// TwinCAT 3 PLC project BX
// ProgramVersion: 3.1.4024.0
// libraries:
//   Tc2_IoFunctions, * (Beckhoff Automation GmbH)
//   Tc2_Math, * (Beckhoff Automation GmbH)
//   Tc2_Standard, * (Beckhoff Automation GmbH)
//   Tc2_System, * (Beckhoff Automation GmbH)
//   Tc2_TcpIp, * (Beckhoff Automation GmbH)
//   Tc2_Utilities, * (Beckhoff Automation GmbH)
//   Tc3_Database, * (Beckhoff Automation GmbH)
//   Tc3_DynamicMemory, * (Beckhoff Automation GmbH)
//   Tc3_EventLogger, * (Beckhoff Automation GmbH)
//   Tc3_JsonXml, * (Beckhoff Automation GmbH)
//   Tc3_Module, * (Beckhoff Automation GmbH)
// project tree:
//   DUTs/00/ DUT_HMI_00.TcDUT, DUT_HMI_00_MANUALS.TcDUT
//   DUTs/01/ DUT_HMI_01.TcDUT, DUT_HMI_01_MANUALS.TcDUT
//   DUTs/02/ DUT_HMI_02.TcDUT, DUT_HMI_02_MANUALS.TcDUT
//   DUTs/03/ DUT_HMI_03.TcDUT, DUT_HMI_03_MANUALS.TcDUT
//   DUTs/04/ DUT_HMI_04.TcDUT, DUT_HMI_04_MANUALS.TcDUT
//   DUTs/05/ DUT_HMI_05.TcDUT, DUT_HMI_05_MANUALS.TcDUT
//   DUTs/06/ DUT_HMI_06.TcDUT, DUT_HMI_06_MANUALS.TcDUT
//   DUTs/07/ DUT_HMI_07.TcDUT, DUT_HMI_07_MANUALS.TcDUT
//   DUTs/08/ DUT_HMI_08.TcDUT, DUT_HMI_08_MANUALS.TcDUT
//   DUTs/09/ DUT_HMI_09.TcDUT, DUT_HMI_09_MANUALS.TcDUT
//   DUTs/10/ DUT_HMI_10.TcDUT, DUT_HMI_10_MANUALS.TcDUT
//   DUTs/11/ DUT_HMI_11.TcDUT, DUT_HMI_11_MANUALS.TcDUT
//   DUTs/12/ DUT_HMI_12.TcDUT, DUT_HMI_12_MANUALS.TcDUT
//   DUTs/13/ DUT_HMI_13.TcDUT, DUT_HMI_13_MANUALS.TcDUT
//   DUTs/14/ DUT_HMI_14.TcDUT, DUT_HMI_14_MANUALS.TcDUT
//   DUTs/15/ DUT_HMI_15.TcDUT, DUT_HMI_15_MANUALS.TcDUT
//   DUTs/16/ DUT_HMI_16.TcDUT, DUT_HMI_16_MANUALS.TcDUT
//   DUTs/Database/ DUT_AppendBatchToProductionQueue.TcDUT, DUT_ChangeBatchPositionInProductionQueue.TcDUT, DUT_CMD_ForceCompletedBatch.TcDUT, DUT_CMD_RecoverBatch.TcDUT, DUT_CMD_RestartBatch.TcDUT, DUT_GetBatchHistory.TcDUT, DUT_GetBatchHistoryDetail.TcDUT, DUT_GetBitting.TcDUT, DUT_CheckCutterAlreadyPresentOnDrums.TcDUT, DUT_GetSettingRepositoryByName.TcDUT, DUT_LogModeStateEvent.TcDUT, DUT_stSPAlarm.TcDUT, DUT_UpdateBroachingProfileSettings.TcDUT, DUT_GetProfilesByFamilyName.TcDUT, DUT_UpdateCuttersOnDrum.TcDUT, DUT_GetResourcesByName.TcDUT, DUT_GetCuttersOnDrum.TcDUT, DUT_NextPartPLCData.TcDUT, DUT_OutInfoOrigin.TcDUT, DUT_ProcessingDataForHMI.TcDUT, DUT_ResourcesByType.TcDUT, DUT_SequenceByName.TcDUT, DUT_SetResourcesByName.TcDUT, DUT_stBroachingPlanBase.TcDUT, DUT_stBatchList.TcDUT, DUT_stBroachingPlanVariants.TcDUT, DUT_stDeleteBatchToProductionQueue.TcDUT, DUT_stExternMarkingData.TcDUT, DUT_stGetPLCData_Buffer.TcDUT, DUT_stMarkingData.TcDUT, DUT_stBroachingPlan.TcDUT, DUT_stOrder.TcDUT, DUT_stOrderItems.TcDUT, DUT_stPLCData.TcDUT, DUT_stProcessingData.TcDUT, DUT_stProcessingHMIData1.TcDUT, DUT_stProcessingHMIData2.TcDUT, DUT_stUpdateBatchToProductionQueue.TcDUT, DUT_UpdateCutterData.TcDUT, DUT_UpdatePartLocationsAndProcessingData.TcDUT, DUT_UpdateSettingRepositoryByName.TcDUT, eDbPiecesStatus.TcDUT
//   DUTs/Database/Mes/ DUT_stMesOrder.TcDUT, DUT_stMesOrderItems.TcDUT
//   DUTs/ DUT_RobSetpoint_Real.TcDUT, DUT_XYZ_Real.TcDUT, DUT_XYZ_Int.TcDUT, eDeviceType.TcTLEO, eLoadingMode.TcDUT, DUT_Events.TcDUT, eBroach.TcDUT, DUT_DataRequest.TcDUT, DUT_MachineData.TcDUT, DUT_MATDiagnostics.TcDUT, DUT_St0Data.TcDUT, DUT_StationData.TcDUT, eConnectionSteps.TcDUT, eEV_Status.TcDUT, eHeaderPieces.TcTLEO, eIcon.TcTLEO, eMode.TcDUT, eProductStatus.TcDUT, eShiftPosMan.TcDUT, eShiftPosPC100.TcDUT, eState.TcTLEO, eStationData.TcDUT, eStationState.TcDUT, stBit.TcDUT, stByteAsBit.TcDUT, stTestStringUnion.TcDUT, stFanucCNCKeyboard.TcDUT, stShiftData.TcDUT, DataBuffer.TcDUT
//   DUTs/EventsMgt/ ST_EventClassInfo.TcDUT, ST_FanucCNCEventAxesMask.TcDUT, ST_FanucCNCEventDetails.TcDUT, ST_FanucCNCEventEntryDetails.TcDUT, ST_FanucCNCEventSourceDetails.TcDUT, ST_FanucCNCEventSourceInfo.TcDUT, ST_FanucCNCEventSourceList.TcDUT, ST_FanucSourceDescriptor.TcDUT, U_FanucCNCEventEntry.TcDUT, U_FanucCNCEventInfo.TcDUT, U_FanucCNCEventSourceInfo.TcDUT
//   DUTs/HMI/ DUT_HIM_ProscessingData.TcDUT, DUT_HIM_DeviceType.TcDUT, DUT_HMI_Display.TcDUT, DUT_HMI_Events.TcDUT, DUT_HMI_EV_Diagnostic.TcDUT, DUT_HMI_EV_Info.TcDUT, DUT_HMI_General.TcDUT, DUT_HMI_General_Manuals.TcDUT, DUT_HMI_Header.TcDUT, DUT_HMI_In.TcDUT, DUT_HMI_In_Resource.TcDUT, DUT_HMI_MesManual.TcDUT, DUT_HMI_Navigation.TcDUT, DUT_HIM_Probe.TcDUT, DUT_HMI_Out.TcDUT, DUT_HMI_Out_Resource.TcDUT, DUT_HMI_Production_Counters.TcDUT, DUT_HMI_Tools.TcDUT, DUT_HMI_UPSStatus.TcDUT
//   DUTs/Production/ DUT_Production.TcDUT, DUT_Production_Counters.TcDUT, DUT_Production_OEE.TcDUT, DUT_Statistics.TcDUT, eOEE.TcDUT
//   FBs/ BytesToWString.TcPOU, FB_ButtonTrigger.TcPOU, FB_DoublingTrigger.TcPOU, FB_LoadingModeChange.TcPOU, FB_OvrMng.TcPOU, FB_PartDataManager.TcPOU, FB_DataBufferManager.TcPOU, FB_PneumaticActuator_2EV.TcPOU, FB_PneumaticActuator_2EV_Diagnostic.TcPOU, FB_Refresh.TcPOU, FB_KillMultipleNavigationPS.TcPOU, FB_RetainTimer.TcPOU, FB_TriggerSequencer.TcPOU, FB_WriteTestFile.TcPOU
//   FBs/Database/FB/ FB_MSSQL_spAppendBatchToProductionQueueFromHMI.TcPOU, FB_MSSQL_spChangeBatchPositionInProductionQueue.TcPOU, FB_MSSQL_spCMD_ForceCompletedBatch.TcPOU, FB_MSSQL_spCMD_HoldBatch.TcPOU, FB_MSSQL_spCMD_RecoverBatch.TcPOU, FB_MSSQL_spCMD_RestartBatch.TcPOU, FB_MSSQL_spCMD_ResumeBatch.TcPOU, FB_MSSQL_spCMD_SuspendBatch.TcPOU, FB_MSSQL_spCMD_UnholdBatch.TcPOU, FB_MSSQL_spDeleteBatchToProductionQueue.TcPOU, FB_MSSQL_spAddProfile.TcPOU, FB_MSSQL_spDeleteCutter.TcPOU, FB_MSSQL_spAddCutter.TcPOU, FB_MSSQL_spGetBatchDetailById.TcPOU, FB_MSSQL_spGetBatchHistory.TcPOU, FB_MSSQL_spGetBatchHistoryByStatus.TcPOU, FB_MSSQL_spGetBatchHistoryDetail.TcPOU, FB_MSSQL_spGetBatchList.TcPOU, FB_MSSQL_spGetBlankKey.TcPOU, FB_MSSQL_spGetBlankKeyByName.TcPOU, FB_MSSQL_spCheckCutterAlreadyPresentOnDrums.TcPOU, FB_MSSQL_spGetCuttersComboboxFormatted.TcPOU, FB_MSSQL_spGetCuttersFromFamilyName.TcPOU, FB_MSSQL_spDeleteProfile.TcPOU, FB_MSSQL_spGetBroachingProfileSettings.TcPOU, FB_MSSQL_spGetSettingRepositoryByName.TcPOU, FB_MSSQL_spUpdateBroachingProfileSettings.TcPOU, FB_MSSQL_spGetProfilesByFamilyName.TcPOU, FB_MSSQL_spGetProfiles.TcPOU, FB_MSSQL_spGetCuttersOnDrum.TcPOU, FB_MSSQL_spGetFamilyNamesForCombobox.TcPOU, FB_MSSQL_spUpdateCuttersOnDrum.TcPOU, FB_MSSQL_spGetCuttersByName.TcPOU, FB_MSSQL_spGetCuttersBySide.TcPOU, FB_MSSQL_spGetCutters.TcPOU, FB_MSSQL_spGetFormattedTablesFromSequences.TcPOU, FB_MSSQL_spGetMillings.TcPOU, FB_MSSQL_spGetMillingsByFamilyName.TcPOU, FB_MSSQL_spGetMillingsByName.TcPOU, FB_MSSQL_spGetOrderInfoList.TcPOU, FB_MSSQL_spGetOrderItems.TcPOU, FB_MSSQL_spGetOrigins.TcPOU, FB_MSSQL_spGetOriginsByName.TcPOU, FB_MSSQL_spGetOriginsBySide.TcPOU, FB_MSSQL_spGetOriginsFromSequence.TcPOU, FB_MSSQL_spGetPartHistory.TcPOU, FB_MSSQL_spGetPartHistoryByBatchName.TcPOU, FB_MSSQL_spGetResourcesByName.TcPOU, FB_MSSQL_spGetResourcesByNameMilling.TcPOU, FB_MSSQL_spGetResourcesByType.TcPOU, FB_MSSQL_spGetResourcesListByType.TcPOU, FB_MSSQL_spGetSettingRepositoryList.TcPOU, FB_MSSQL_spGetSideCode.TcPOU, FB_MSSQL_spSetResourcesByName.TcPOU, FB_MSSQL_spUpdateBatchToProductionQueue.TcPOU, FB_MSSQL_spUpdateCutterData.TcPOU, FB_MSSQL_spUpdateSettingRepositoryByName.TcPOU
//   FBs/Database/FB/Mes/ FB_MSSQL_spMES_GetOrderInfoList.TcPOU, FB_MSSQL_spMES_GetOrderItems.TcPOU
//   FBs/Database/ FB_HMI_SP_Alarm.TcPOU, FB_ProcessingData.TcPOU, PRG_MSSQL_InitConnection.TcPOU, PRG_MSSQL_InitConnection_MyTest1.TcPOU, PRG_MSSQL_InitConnection_MyTest2.TcPOU, PRG_MSSQL_InitConnection_MyTest3.TcPOU, PRG_MSSQL_InitConnection_MyTest4.TcPOU, PRG_MSSQL_InitConnection_MyTest5.TcPOU, PRG_MSSQL_spCMD_AbortProduction.TcPOU, PRG_MSSQL_spMyTest.TcPOU, PRG_MSSQL_spLogModeStateEvent.TcPOU, PRG_MSSQL_spGetNextPartPLCData.TcPOU, PRG_MSSQL_spGetProcessingDataForHMI.TcPOU, PRG_MSSQL_UpdatePartLocationsAndProcessingData.TcPOU
//   FBs/DataRequest/ FB_DataRequest.TcPOU, FC_UnloadManager.TcPOU, FC_BroachingPlanCopyPass.TcPOU, FC_BroachingPlanCopyConpensation.TcPOU, FC_DataFind.TcPOU
//   FBs/Ethernet/ FB_ClientConnection.TcPOU, FB_EthDevice.TcPOU, FB_FrameFifo.TcPOU
//   FBs/Events/ FB_CheckFanucCNCActiveEvents.TcPOU, FB_CheckFanucPMCActiveEvents.TcPOU, FB_PMCEventCollectors.TcPOU, I_EventDetailer.TcIO
//   FBs/LaserMarker - LASIT/ DUT_Job.TcDUT, FB_FlyPowerMarkExeManager.TcPOU, FB_Lasit.TcPOU, FB_LasitManager.TcPOU, FB_FlyPowerMarkManager.TcPOU, FC_Check_ACK.TcPOU, FC_Check_EOT.TcPOU, FC_Check_IN.TcPOU, FC_Check_J.TcPOU, FC_Check_K.TcPOU, FC_Check_R.TcPOU, FC_Check_S.TcPOU, FC_Check_SOH.TcPOU, FC_Check_STX.TcPOU, FC_Check_T.TcPOU
//   FBs/StringBuilder/ clsStringBuilder.TcPOU, I_LimitedStringBuilder.TcIO, I_StringBuilder.TcIO
//   FCs/ FC_AlarmExists.TcPOU, FC_BYTE_TO_BOOLARR.TcPOU, FC_BOOLARR_TO_BYTE.TcPOU, FC_BOOLBYTE_TO_BYTE.TcPOU, FC_BYTE_TO_BOOLBYTE.TcPOU, FC_Concat4.TcPOU, FC_CycleTimeToString.TcPOU, FC_DT_TO_ISO8610.TcPOU, FC_EnumSnakeCaseToString.TcPOU, FC_HeaderCounters.TcPOU, FC_MarkingLayoutSelection.TcPOU, FC_myDTtoString.TcPOU, FC_UpdatePieceCount.TcPOU, FC_OvrManagement.TcPOU, FC_PMCAlarmToBoolArray.TcPOU, FC_PMCWarningToBoolArray.TcPOU, FC_ProductStatus.TcPOU, FC_ProductStatusDatabase.TcPOU, FC_ProductStatusNoPresence.TcPOU, FC_OeeSetUpdateCount.TcPOU, FC_SetPartProgramNameByID.TcPOU, FC_ToBoolArray.TcPOU, FC_ToByte.TcPOU, FC_WIDP_TO_PPNAME.TcPOU, Inc.TcPOU, Print.TcPOU
//   GVLs/ CNC.TcGVL, DB.TcGVL, EC.TcGVL, ETH.TcGVL, G.TcGVL, HMI.TcGVL
//   / PlcTask.TcTTO, ServiceTask.TcTTO
//   POUs/ Database.TcPOU, MAIN.TcPOU, MAIN_SERVICE.TcPOU, PF_00_UPS.TcPOU, PRG_Diagnostic.TcPOU, PRG_EventManagement.TcPOU, PRG_OEE.TcPOU
// real-time tasks:
//   TASK PlcTask: cycle T#1ms, priority 4, ADS port 350
//   TASK ServiceTask: cycle T#50000us, priority 8, ADS port 351
// I/O:
//   DEVICE LAN 1 (EtherCAT), AmsNetId 192.168.159.1.2.1
//     A651 (EP5151-0002) [EP5151-0002 1Ch. Inc. Encoder 24V, M12, single ended]
//     AL671 (CTEU-EtherCAT Modular) [CTEU-EtherCAT Fieldbus modular]
//       modules: Module 1 (VAEM-L1-S-24-PT [48DO])
//     AL673 (CTEU-EtherCAT Modular) [CTEU-EtherCAT Fieldbus modular]
//       modules: Module 1 (VAEM-L1-S-24-PT [48DO])
//   DEVICE LAN 2 (Profinet Device), AmsNetId 192.168.2.200.3.1
//     tcpniodevice [Beckhoff Automation TwinCAT PLC PROFINET I/O Device with I/Os, V2.32, 1 port TwinCAT PN Device]
//       modules: Term 1 (DAP Module), X400 (100 Byte Input), R2000 (200 Byte Input), D2000 (200 Byte Input), Y400 (100 Byte Output), R2200 (200 Byte Output), D2200 (200 Byte Output)
// variable links:
//   BX/BX Instance <-> LAN 1 (EtherCAT)
//     ServiceTask Inputs/EC.EtherCAT_DevState <-> Inputs/DevState
//   BX/BX Instance <-> LAN 1 (EtherCAT)/A651 (EP5151-0002)
//     PlcTask Inputs/EC.I_Ovr_CounterValue <-> ENC Status compact/Counter value
//     PlcTask Inputs/EC.I_Ovr_Overflow <-> ENC Status compact/Status/Counter overflow
//     PlcTask Inputs/EC.I_Ovr_SetCounterDone <-> ENC Status compact/Status/Set counter done
//     PlcTask Inputs/EC.I_Ovr_Underflow <-> ENC Status compact/Status/Counter underflow
//     PlcTask Outputs/EC.Q_Ovr_SetCounter <-> ENC Control compact/Control/Set counter
//     PlcTask Outputs/EC.Q_Ovr_SetCounterValue <-> ENC Control compact/Set counter value
//   BX/BX Instance <-> LAN 1 (EtherCAT)/AL671 (CTEU-EtherCAT Modular)
//     PlcTask Outputs/EC.AL671[{0..4}] <-> Module 1 (VAEM-L1-S-24-PT [48DO])/Outputs/C{1..5} Output  (5 links)
//   BX/BX Instance <-> LAN 1 (EtherCAT)/AL673 (CTEU-EtherCAT Modular)
//     PlcTask Outputs/EC.AL673[{0..5}] <-> Module 1 (VAEM-L1-S-24-PT [48DO])/Outputs/C{1..6} Output  (6 links)
//   BX/BX Instance <-> LAN 2 (Profinet Device)
//     ServiceTask Inputs/EC.ProfiNET_DevState <-> Inputs/DevState
//   BX/BX Instance <-> LAN 2 (Profinet Device)/tcpniodevice
//     PlcTask Inputs/CNC.I_D2200 <-> API/D2200 (200 Byte Output)/Subterm 9 (200 Byte Output)/Inputs/1 Byte Output[0]
//     PlcTask Inputs/CNC.I_D2200 @bit {8..1592 step 8} <-> API/D2200 (200 Byte Output)/Subterm 9 (200 Byte Output)/Inputs/1 Byte Output[{1..199}]  (199 links)
//     PlcTask Inputs/CNC.I_R2200 <-> API/R2200 (200 Byte Output)/Subterm 8 (200 Byte Output)/Inputs/1 Byte Output[0]
//     PlcTask Inputs/CNC.I_R2200 @bit {8..1592 step 8} <-> API/R2200 (200 Byte Output)/Subterm 8 (200 Byte Output)/Inputs/1 Byte Output[{1..199}]  (199 links)
//     PlcTask Inputs/CNC.I_Y400 <-> API/Y400 (100 Byte Output)/Subterm 7 (100 Byte Output)/Inputs/1 Byte Output[0]
//     PlcTask Inputs/CNC.I_Y400 @bit {8..792 step 8} <-> API/Y400 (100 Byte Output)/Subterm 7 (100 Byte Output)/Inputs/1 Byte Output[{1..99}]  (99 links)
//     PlcTask Outputs/CNC.Q_D2000 <-> API/D2000 (200 Byte Input)/Subterm 6 (200 Byte Input)/Outputs/1 Byte Input[0]
//     PlcTask Outputs/CNC.Q_D2000 @bit {8..1592 step 8} <-> API/D2000 (200 Byte Input)/Subterm 6 (200 Byte Input)/Outputs/1 Byte Input[{1..199}]  (199 links)
//     PlcTask Outputs/CNC.Q_R2000 <-> API/R2000 (200 Byte Input)/Subterm 5 (200 Byte Input)/Outputs/1 Byte Input[0]
//     PlcTask Outputs/CNC.Q_R2000 @bit {8..1592 step 8} <-> API/R2000 (200 Byte Input)/Subterm 5 (200 Byte Input)/Outputs/1 Byte Input[{1..199}]  (199 links)
//     ServiceTask Outputs/CNC.Q_X400 <-> API/X400 (100 Byte Input)/Subterm 4 (100 Byte Input)/Outputs/1 Byte Input[0]
//     ServiceTask Outputs/CNC.Q_X400 @bit {8..792 step 8} <-> API/X400 (100 Byte Input)/Subterm 4 (100 Byte Input)/Outputs/1 Byte Input[{1..99}]  (99 links)

CONFIGURATION BX
    RESOURCE PLC ON TwinCAT3
        TASK PlcTask(INTERVAL := T#1ms, PRIORITY := 4);
        TASK ServiceTask(INTERVAL := T#50000us, PRIORITY := 8);
        PROGRAM MAIN WITH PlcTask : MAIN;
        PROGRAM MAIN_SERVICE WITH ServiceTask : MAIN_SERVICE;
    END_RESOURCE
END_CONFIGURATION

// ---- DUTs/00/DUT_HMI_00.TcDUT
TYPE DUT_HMI_00 :
STRUCT
	Manuals 		: DUT_HMI_00_MANUALS;
	EVDiagnostic 	: ARRAY[3..47] OF DUT_HMI_EV_Diagnostic;
	EVInfo			: ARRAY[0..CNC.NUM_MAX_MANUALS_00-1] OF DUT_HMI_EV_Info;
	Status			: USINT;
	CycleTime		: STRING;
END_STRUCT
END_TYPE

// ---- DUTs/00/DUT_HMI_00_MANUALS.TcDUT
TYPE DUT_HMI_00_MANUALS :
STRUCT
	PS : ARRAY[0..CNC.NUM_MAX_MANUALS_00-1] OF BOOL;
	LS : ARRAY[0..CNC.NUM_MAX_MANUALS_00-1] OF BOOL;
END_STRUCT
END_TYPE

// ---- DUTs/01/DUT_HMI_01.TcDUT
TYPE DUT_HMI_01 :
STRUCT
	Manuals 		: DUT_HMI_01_MANUALS;
	ProductStatus 	: eProductStatus;
	State			: eStationState;
	EVDiagnostic 	: ARRAY[0..20] OF DUT_HMI_EV_Diagnostic;
	EVInfo			: ARRAY[0..CNC.NUM_MAX_MANUALS_01-1] OF DUT_HMI_EV_Info;
	Status			: USINT;
	CycleTime		: STRING;
END_STRUCT
END_TYPE

// ---- DUTs/01/DUT_HMI_01_MANUALS.TcDUT
TYPE DUT_HMI_01_MANUALS :
STRUCT
	PS : ARRAY[0..CNC.NUM_MAX_MANUALS_01-1] OF BOOL;
	LS : ARRAY[0..CNC.NUM_MAX_MANUALS_01-1] OF BOOL;
END_STRUCT
END_TYPE

// ---- DUTs/02/DUT_HMI_02.TcDUT
TYPE DUT_HMI_02 :
STRUCT
	Manuals : DUT_HMI_02_MANUALS;
	ProductStatus 	: eProductStatus;
	State			: eStationState;
	EVDiagnostic 	: ARRAY[0..20] OF DUT_HMI_EV_Diagnostic;
	EVInfo			: ARRAY[0..CNC.NUM_MAX_MANUALS_02-1] OF DUT_HMI_EV_Info;
	Status			: USINT;
	CycleTime		: STRING;
END_STRUCT
END_TYPE

// ---- DUTs/02/DUT_HMI_02_MANUALS.TcDUT
TYPE DUT_HMI_02_MANUALS :
STRUCT
	PS : ARRAY[0..CNC.NUM_MAX_MANUALS_02-1] OF BOOL;
	LS : ARRAY[0..CNC.NUM_MAX_MANUALS_02-1] OF BOOL;
END_STRUCT
END_TYPE

// ---- DUTs/03/DUT_HMI_03.TcDUT
TYPE DUT_HMI_03 :
STRUCT
	Manuals : DUT_HMI_03_MANUALS;
	ProductStatus 	: eProductStatus;
	TON_DelayProductStatus : TON;
	RTRIG_ProductStatus : R_TRIG;
	State			: eStationState;
	EVDiagnostic 	: ARRAY[0..20] OF DUT_HMI_EV_Diagnostic;
	EVInfo			: ARRAY[0..CNC.NUM_MAX_MANUALS_03-1] OF DUT_HMI_EV_Info;
	Status			: USINT;
	CycleTime		: STRING;
END_STRUCT
END_TYPE

// ---- DUTs/03/DUT_HMI_03_MANUALS.TcDUT
TYPE DUT_HMI_03_MANUALS :
STRUCT
	PS : ARRAY[0..CNC.NUM_MAX_MANUALS_03-1] OF BOOL;
	LS : ARRAY[0..CNC.NUM_MAX_MANUALS_03-1] OF BOOL;
END_STRUCT
END_TYPE

// ---- DUTs/04/DUT_HMI_04.TcDUT
TYPE DUT_HMI_04 :
STRUCT
	Manuals : DUT_HMI_04_MANUALS;
	ProductStatus 	: eProductStatus;
	State			: eStationState;
	EVDiagnostic 	: ARRAY[0..20] OF DUT_HMI_EV_Diagnostic;
	EVInfo			: ARRAY[0..CNC.NUM_MAX_MANUALS_04-1] OF DUT_HMI_EV_Info;
	Status			: USINT;
	CycleTime		: STRING;
	BroachTarget	: USINT;
END_STRUCT
END_TYPE

// ---- DUTs/04/DUT_HMI_04_MANUALS.TcDUT
TYPE DUT_HMI_04_MANUALS :
STRUCT
	PS : ARRAY[0..CNC.NUM_MAX_MANUALS_04-1] OF BOOL;
	LS : ARRAY[0..CNC.NUM_MAX_MANUALS_04-1] OF BOOL;
END_STRUCT
END_TYPE

// ---- DUTs/05/DUT_HMI_05.TcDUT
TYPE DUT_HMI_05 :
STRUCT
	Manuals : DUT_HMI_05_MANUALS;
	ProductStatus 	: eProductStatus;
	State			: eStationState;
	EVDiagnostic 	: ARRAY[0..20] OF DUT_HMI_EV_Diagnostic;
	EVInfo			: ARRAY[0..CNC.NUM_MAX_MANUALS_05-1] OF DUT_HMI_EV_Info;
	Status			: USINT;
	CycleTime		: STRING;
	BroachTarget	: USINT;
END_STRUCT
END_TYPE

// ---- DUTs/05/DUT_HMI_05_MANUALS.TcDUT
TYPE DUT_HMI_05_MANUALS :
STRUCT
	PS : ARRAY[0..CNC.NUM_MAX_MANUALS_05-1] OF BOOL;
	LS : ARRAY[0..CNC.NUM_MAX_MANUALS_05-1] OF BOOL;
END_STRUCT
END_TYPE

// ---- DUTs/06/DUT_HMI_06.TcDUT
TYPE DUT_HMI_06 :
STRUCT
	Manuals : DUT_HMI_06_MANUALS;
	ProductStatus 	: eProductStatus;
	State			: eStationState;
	EVDiagnostic 	: ARRAY[0..20] OF DUT_HMI_EV_Diagnostic;
	EVInfo			: ARRAY[0..CNC.NUM_MAX_MANUALS_06-1] OF DUT_HMI_EV_Info;
	Status			: USINT;
	CycleTime		: STRING;
	BroachTarget	: USINT;
END_STRUCT
END_TYPE

// ---- DUTs/06/DUT_HMI_06_MANUALS.TcDUT
TYPE DUT_HMI_06_MANUALS :
STRUCT
	PS : ARRAY[0..CNC.NUM_MAX_MANUALS_06-1] OF BOOL;
	LS : ARRAY[0..CNC.NUM_MAX_MANUALS_06-1] OF BOOL;
END_STRUCT
END_TYPE

// ---- DUTs/07/DUT_HMI_07.TcDUT
TYPE DUT_HMI_07 :
STRUCT
	Manuals : DUT_HMI_07_MANUALS;
	ProductStatus 	: eProductStatus;
	State			: eStationState;
	EVDiagnostic 	: ARRAY[0..20] OF DUT_HMI_EV_Diagnostic;
	EVInfo			: ARRAY[0..CNC.NUM_MAX_MANUALS_07-1] OF DUT_HMI_EV_Info;
	Status			: USINT;
	CycleTime		: STRING;
	BroachTarget	: USINT;
END_STRUCT
END_TYPE

// ---- DUTs/07/DUT_HMI_07_MANUALS.TcDUT
TYPE DUT_HMI_07_MANUALS :
STRUCT
	PS : ARRAY[0..CNC.NUM_MAX_MANUALS_07-1] OF BOOL;
	LS : ARRAY[0..CNC.NUM_MAX_MANUALS_07-1] OF BOOL;
END_STRUCT
END_TYPE

// ---- DUTs/08/DUT_HMI_08.TcDUT
TYPE DUT_HMI_08 :
STRUCT
	Manuals : DUT_HMI_08_MANUALS;
	ProductStatus 	: eProductStatus;
	State			: eStationState;
	EVDiagnostic 	: ARRAY[0..20] OF DUT_HMI_EV_Diagnostic;
	EVInfo			: ARRAY[0..CNC.NUM_MAX_MANUALS_08-1] OF DUT_HMI_EV_Info;
	Status			: USINT;
	CycleTime		: STRING;
	BroachTarget	: USINT;
END_STRUCT
END_TYPE

// ---- DUTs/08/DUT_HMI_08_MANUALS.TcDUT
TYPE DUT_HMI_08_MANUALS :
STRUCT
	PS : ARRAY[0..CNC.NUM_MAX_MANUALS_08-1] OF BOOL;
	LS : ARRAY[0..CNC.NUM_MAX_MANUALS_08-1] OF BOOL;
END_STRUCT
END_TYPE

// ---- DUTs/09/DUT_HMI_09.TcDUT
TYPE DUT_HMI_09 :
STRUCT
	Manuals : DUT_HMI_09_MANUALS;
	ProductStatus 	: eProductStatus;
	TON_DelayProductStatus : TON;
	RTRIG_ProductStatus : R_TRIG;
	State			: eStationState;
	EVDiagnostic 	: ARRAY[0..20] OF DUT_HMI_EV_Diagnostic;
	EVInfo			: ARRAY[0..CNC.NUM_MAX_MANUALS_09-1] OF DUT_HMI_EV_Info;
	Status			: USINT;
	CycleTime		: STRING;
	BroachTarget	: USINT;
END_STRUCT
END_TYPE

// ---- DUTs/09/DUT_HMI_09_MANUALS.TcDUT
TYPE DUT_HMI_09_MANUALS :
STRUCT
	PS : ARRAY[0..CNC.NUM_MAX_MANUALS_09-1] OF BOOL;
	LS : ARRAY[0..CNC.NUM_MAX_MANUALS_09-1] OF BOOL;
END_STRUCT
END_TYPE

// ---- DUTs/10/DUT_HMI_10.TcDUT
TYPE DUT_HMI_10 :
STRUCT
	Manuals : DUT_HMI_10_MANUALS;
	ProductStatus 	: eProductStatus;
	State			: eStationState;
	EVDiagnostic 	: ARRAY[0..20] OF DUT_HMI_EV_Diagnostic;
	EVInfo			: ARRAY[0..CNC.NUM_MAX_MANUALS_10-1] OF DUT_HMI_EV_Info;
	Status			: USINT;
	CycleTime		: STRING;
	BroachTarget	: USINT;
END_STRUCT
END_TYPE

// ---- DUTs/10/DUT_HMI_10_MANUALS.TcDUT
TYPE DUT_HMI_10_MANUALS :
STRUCT
	PS : ARRAY[0..CNC.NUM_MAX_MANUALS_10-1] OF BOOL;
	LS : ARRAY[0..CNC.NUM_MAX_MANUALS_10-1] OF BOOL;
END_STRUCT
END_TYPE

// ---- DUTs/11/DUT_HMI_11.TcDUT
TYPE DUT_HMI_11 :
STRUCT
	Manuals : DUT_HMI_11_MANUALS;
	ProductStatus 	: eProductStatus;
	State			: eStationState;
	EVDiagnostic 	: ARRAY[0..20] OF DUT_HMI_EV_Diagnostic;
	EVInfo			: ARRAY[0..CNC.NUM_MAX_MANUALS_11-1] OF DUT_HMI_EV_Info;
	Status			: USINT;
	CycleTime		: STRING;
END_STRUCT
END_TYPE

// ---- DUTs/11/DUT_HMI_11_MANUALS.TcDUT
TYPE DUT_HMI_11_MANUALS :
STRUCT
	PS : ARRAY[0..CNC.NUM_MAX_MANUALS_11-1] OF BOOL;
	LS : ARRAY[0..CNC.NUM_MAX_MANUALS_11-1] OF BOOL;
END_STRUCT
END_TYPE

// ---- DUTs/12/DUT_HMI_12.TcDUT
TYPE DUT_HMI_12 :
STRUCT
	Manuals : DUT_HMI_12_MANUALS;
	ProductStatus 	: eProductStatus;
	State			: eStationState;
	EVDiagnostic 	: ARRAY[0..20] OF DUT_HMI_EV_Diagnostic;
	EVInfo			: ARRAY[0..CNC.NUM_MAX_MANUALS_12-1] OF DUT_HMI_EV_Info;
	Status			: USINT;
	CycleTime		: STRING;
END_STRUCT
END_TYPE

// ---- DUTs/12/DUT_HMI_12_MANUALS.TcDUT
TYPE DUT_HMI_12_MANUALS :
STRUCT
	PS : ARRAY[0..CNC.NUM_MAX_MANUALS_12-1] OF BOOL;
	LS : ARRAY[0..CNC.NUM_MAX_MANUALS_12-1] OF BOOL;
END_STRUCT
END_TYPE

// ---- DUTs/13/DUT_HMI_13.TcDUT
TYPE DUT_HMI_13 :
STRUCT
	Manuals : DUT_HMI_13_MANUALS;
	ProductStatus 	: eProductStatus;
	State			: eStationState;
	EVDiagnostic 	: ARRAY[0..20] OF DUT_HMI_EV_Diagnostic;
	EVInfo			: ARRAY[0..CNC.NUM_MAX_MANUALS_13-1] OF DUT_HMI_EV_Info;
	Status			: USINT;
	CycleTime		: STRING;
END_STRUCT
END_TYPE

// ---- DUTs/13/DUT_HMI_13_MANUALS.TcDUT
TYPE DUT_HMI_13_MANUALS :
STRUCT
	PS : ARRAY[0..CNC.NUM_MAX_MANUALS_13-1] OF BOOL;
	LS : ARRAY[0..CNC.NUM_MAX_MANUALS_13-1] OF BOOL;
END_STRUCT
END_TYPE

// ---- DUTs/14/DUT_HMI_14.TcDUT
TYPE DUT_HMI_14 :
STRUCT
	Manuals : DUT_HMI_14_MANUALS;
	ProductStatus 	: eProductStatus;
	State			: eStationState;
	EVDiagnostic 	: ARRAY[0..20] OF DUT_HMI_EV_Diagnostic;
	EVInfo			: ARRAY[0..CNC.NUM_MAX_MANUALS_14-1] OF DUT_HMI_EV_Info;
	Status			: USINT;
	CycleTime		: STRING;
END_STRUCT
END_TYPE

// ---- DUTs/14/DUT_HMI_14_MANUALS.TcDUT
TYPE DUT_HMI_14_MANUALS :
STRUCT
	PS : ARRAY[0..CNC.NUM_MAX_MANUALS_14-1] OF BOOL;
	LS : ARRAY[0..CNC.NUM_MAX_MANUALS_14-1] OF BOOL;
END_STRUCT
END_TYPE

// ---- DUTs/15/DUT_HMI_15.TcDUT
TYPE DUT_HMI_15 :
STRUCT
	Manuals : DUT_HMI_15_MANUALS;
	ProductStatus 	: eProductStatus;
	State			: eStationState;
	EVDiagnostic 	: ARRAY[0..20] OF DUT_HMI_EV_Diagnostic;
	EVInfo			: ARRAY[0..CNC.NUM_MAX_MANUALS_15-1] OF DUT_HMI_EV_Info;
	Status			: USINT;
	CycleTime		: STRING;
END_STRUCT
END_TYPE

// ---- DUTs/15/DUT_HMI_15_MANUALS.TcDUT
TYPE DUT_HMI_15_MANUALS :
STRUCT
	PS : ARRAY[0..CNC.NUM_MAX_MANUALS_15-1] OF BOOL;
	LS : ARRAY[0..CNC.NUM_MAX_MANUALS_15-1] OF BOOL;
END_STRUCT
END_TYPE

// ---- DUTs/16/DUT_HMI_16.TcDUT
TYPE DUT_HMI_16 :
STRUCT
	Manuals : DUT_HMI_16_MANUALS;
	ProductStatus 	: eProductStatus;
	State			: eStationState;
	EVDiagnostic 	: ARRAY[0..20] OF DUT_HMI_EV_Diagnostic;
	EVInfo			: ARRAY[0..CNC.NUM_MAX_MANUALS_16-1] OF DUT_HMI_EV_Info;
	Status			: USINT;
	CycleTime		: STRING;
END_STRUCT
END_TYPE

// ---- DUTs/16/DUT_HMI_16_MANUALS.TcDUT
TYPE DUT_HMI_16_MANUALS :
STRUCT
	PS : ARRAY[0..CNC.NUM_MAX_MANUALS_16-1] OF BOOL;
	LS : ARRAY[0..CNC.NUM_MAX_MANUALS_16-1] OF BOOL;
END_STRUCT
END_TYPE

// ---- DUTs/Database/DUT_AppendBatchToProductionQueue.TcDUT
TYPE DUT_AppendBatchToProductionQueue :
STRUCT
	return_					: DINT;
	BatchInfoJson			: STRING(DB.MAX_STRING_SIZE);
	BatchItemsJson			: STRING(DB.MAX_STRING_SIZE);
END_STRUCT
END_TYPE

// ---- DUTs/Database/DUT_ChangeBatchPositionInProductionQueue.TcDUT
TYPE DUT_ChangeBatchPositionInProductionQueue:
STRUCT  
	return_value		: DINT;
	BatchId				: STRING(50);
	DestinationPosition : DINT;
END_STRUCT
END_TYPE

// ---- DUTs/Database/DUT_CMD_ForceCompletedBatch.TcDUT
TYPE DUT_CMD_ForceCompletedBatch:
STRUCT  
	return_value	: DINT;
	Id	: STRING(50);
END_STRUCT
END_TYPE

// ---- DUTs/Database/DUT_CMD_RecoverBatch.TcDUT
TYPE DUT_CMD_RecoverBatch:
STRUCT  
	return_value	: DINT;
	Id	: STRING(50);
	Mode	: STRING(50);
END_STRUCT
END_TYPE

// ---- DUTs/Database/DUT_CMD_RestartBatch.TcDUT
TYPE DUT_CMD_RestartBatch:
STRUCT  
	return_value	: DINT;
	Id	: STRING(50);
	Mode	: STRING(50);
	RestartMode	: STRING(50);
END_STRUCT
END_TYPE

// ---- DUTs/Database/DUT_GetBatchHistory.TcDUT
TYPE DUT_GetBatchHistory:
STRUCT  
	return_value	: DINT;
	CurrentPage	: DINT;
	RecordToFetch	: DINT;
END_STRUCT
END_TYPE

// ---- DUTs/Database/DUT_GetBatchHistoryDetail.TcDUT
TYPE DUT_GetBatchHistoryDetail:
STRUCT  
	return_value	: DINT;
	BatchId			: STRING(50);
END_STRUCT
END_TYPE

// ---- DUTs/Database/DUT_GetBitting.TcDUT
TYPE DUT_GetBitting :
STRUCT
	CodeSchema				: STRING(50);
	SideBar					: STRING(50);
END_STRUCT
END_TYPE

// ---- DUTs/Database/DUT_CheckCutterAlreadyPresentOnDrums.TcDUT
TYPE DUT_CheckCutterAlreadyPresentOnDrums :
STRUCT
	Id			: DINT;
	Drum		: STRING(30);
	Present		: DINT;
END_STRUCT
END_TYPE

// ---- DUTs/Database/DUT_GetSettingRepositoryByName.TcDUT
TYPE DUT_GetSettingRepositoryByName:
STRUCT  
	Name		: STRING(50);
	Data		: STRING(DB.MAX_STRING_SIZE);
END_STRUCT
END_TYPE

// ---- DUTs/Database/DUT_LogModeStateEvent.TcDUT
TYPE DUT_LogModeStateEvent :
STRUCT
	return_value 	: DINT;
	EventId			: LINT;
	EventTimeStamp  : DT;
	EventType       : DINT;
	Mode            : DINT;
	State           : DINT;
END_STRUCT
END_TYPE

// ---- DUTs/Database/DUT_stSPAlarm.TcDUT
TYPE DUT_stSPAlarm :
STRUCT
	Error : BOOL;
	ErrorID : DINT;
END_STRUCT
END_TYPE

// ---- DUTs/Database/DUT_UpdateBroachingProfileSettings.TcDUT
TYPE DUT_UpdateBroachingProfileSettings :
STRUCT
	IdBroachingProfileSettings	: DINT;
	DataBroachingProfile		: STRING(DB.MAX_STRING_SIZE);
END_STRUCT
END_TYPE

// ---- DUTs/Database/DUT_GetProfilesByFamilyName.TcDUT
TYPE DUT_GetProfilesByFamilyName :
STRUCT
	FamilyName		: STRING(30);
	JsonResult	: STRING(DB.MAX_STRING_SIZE);
END_STRUCT
END_TYPE

// ---- DUTs/Database/DUT_UpdateCuttersOnDrum.TcDUT
TYPE DUT_UpdateCuttersOnDrum :
STRUCT
	Drum		: STRING(30);
	JsonValue	: STRING(DB.MAX_STRING_SIZE);
END_STRUCT
END_TYPE

// ---- DUTs/Database/DUT_GetResourcesByName.TcDUT
TYPE DUT_GetResourcesByName :
STRUCT
	return_value	: DINT;
	ResourceName	: STRING(50);
END_STRUCT
END_TYPE

// ---- DUTs/Database/DUT_GetCuttersOnDrum.TcDUT
TYPE DUT_GetCuttersOnDrum :
STRUCT
	Drum		: STRING(30);
	JsonResult	: STRING(DB.MAX_STRING_SIZE);
END_STRUCT
END_TYPE

// ---- DUTs/Database/DUT_NextPartPLCData.TcDUT
TYPE DUT_NextPartPLCData :
STRUCT
	return_value: DINT;
	PLCData : STRING(DB.MAX_STRING_SIZE);
END_STRUCT
END_TYPE

// ---- DUTs/Database/DUT_OutInfoOrigin.TcDUT
TYPE DUT_OutInfoOrigin :
STRUCT
	OriginName		: STRING(50);
	NameX			: STRING(10);
	X				: REAL;
	NameY			: STRING(10);
	Y				: REAL;
	NameZ			: STRING(10);
	Z				: REAL;
	NameB			: STRING(10);
	B				: REAL;
END_STRUCT
END_TYPE

// ---- DUTs/Database/DUT_ProcessingDataForHMI.TcDUT
TYPE DUT_ProcessingDataForHMI :
STRUCT
	return_: DINT;
	ProcessingData : STRING(DB.MAX_STRING_SIZE);
END_STRUCT
END_TYPE

// ---- DUTs/Database/DUT_ResourcesByType.TcDUT
TYPE DUT_ResourcesByType :
STRUCT
	return_value	: DINT;
	ReaourceType	: STRING(50);
END_STRUCT
END_TYPE

// ---- DUTs/Database/DUT_SequenceByName.TcDUT
TYPE DUT_SequenceByName :
STRUCT
	return_value	: DINT;
	SequenceName	: STRING(50);
END_STRUCT
END_TYPE

// ---- DUTs/Database/DUT_SetResourcesByName.TcDUT
TYPE DUT_SetResourcesByName :
STRUCT
	return_value	: DINT;
	ReaourceName	: STRING(50);
	NewData			: STRING(DB.MAX_STRING_SIZE);
END_STRUCT
END_TYPE

// ---- DUTs/Database/DUT_stBroachingPlanBase.TcDUT
TYPE DUT_stBroachingPlanBase :
STRUCT
	ToolHolderBase_Position 				: DINT;
	ToolHolderBase_BroachName 			: STRING(50);
	ToolHolderBase_LateralCompensation 	: REAL;
	ToolHolderBase_DepthCompensation 	: REAL;
	ToolHolderBase_AngleCompensation 	: REAL;
END_STRUCT
END_TYPE

// ---- DUTs/Database/DUT_stBatchList.TcDUT
TYPE DUT_stBatchList :
STRUCT
	return_			: DINT;
	InputJson	: STRING(DB.MAX_STRING_SIZE);
	OutputJson	: STRING(DB.MAX_STRING_SIZE);
END_STRUCT
END_TYPE

// ---- DUTs/Database/DUT_stBroachingPlanVariants.TcDUT
TYPE DUT_stBroachingPlanVariants :
STRUCT
   ToolHolderA_Position				: DINT;
   ToolHolderA_BroachName			: STRING(50);
   ToolHolderA_LateralCompensation	: REAL;
   ToolHolderA_DepthCompensation	: REAL;
   ToolHolderA_AngleCompensation	: REAL;
   ToolHolderB_Position				: DINT;
   ToolHolderB_BroachName			: STRING(50);
   ToolHolderB_LateralCompensation	: REAL;
   ToolHolderB_DepthCompensation	: REAL;
   ToolHolderB_AngleCompensation	: REAL;
   ToolHolderC_Position				: DINT;
   ToolHolderC_BroachName			: STRING(50);
   ToolHolderC_LateralCompensation	: REAL;
   ToolHolderC_DepthCompensation	: REAL;
   ToolHolderC_AngleCompensation	: REAL;
   ToolHolderD_Position				: DINT;
   ToolHolderD_BroachName			: STRING(50);
   ToolHolderD_LateralCompensation	: REAL;
   ToolHolderD_DepthCompensation	: REAL;
   ToolHolderD_AngleCompensation	: REAL;
   ToolHolderE_Position				: DINT;
   ToolHolderE_BroachName			: STRING(50);
   ToolHolderE_LateralCompensation	: REAL;
   ToolHolderE_DepthCompensation	: REAL;
   ToolHolderE_AngleCompensation	: REAL;
   ToolHolderF_Position				: DINT;
   ToolHolderF_BroachName			: STRING(50);
   ToolHolderF_LateralCompensation	: REAL;
   ToolHolderF_DepthCompensation	: REAL;
   ToolHolderF_AngleCompensation	: REAL;
END_STRUCT
END_TYPE

// ---- DUTs/Database/DUT_stDeleteBatchToProductionQueue.TcDUT
TYPE DUT_stDeleteBatchToProductionQueue :
STRUCT
	return_			: DINT;
	BatchId	: STRING(50);
END_STRUCT
END_TYPE

// ---- DUTs/Database/DUT_stExternMarkingData.TcDUT
TYPE DUT_stExternMarkingData :
STRUCT
	FrontEnable : ARRAY[0..7] OF BOOL;
	FrontText1 	: STRING(50);
	FrontText2 	: STRING(50);
	FrontText3 	: STRING(50);
	FrontText4 	: STRING(50);
	FrontText5 	: STRING(50);
	FrontText6 	: STRING(50);
	BackEnable 	: ARRAY[0..7] OF BOOL;
	BackText1 	: STRING(50);
	BackText2 	: STRING(50);
	BackText3 	: STRING(50);
	BackText4 	: STRING(50);
	BackText5 	: STRING(50);
	BackText6 	: STRING(50);
END_STRUCT
END_TYPE

// ---- DUTs/Database/DUT_stGetPLCData_Buffer.TcDUT
TYPE DUT_stGetPLCData_Buffer :
STRUCT
	PLCData: STRING(DB.MAX_STRING_SIZE);
END_STRUCT
END_TYPE

// ---- DUTs/Database/DUT_stMarkingData.TcDUT
TYPE DUT_stMarkingData :
STRUCT
    LayoutName 		: STRING(50);
    OrderReference 	: STRING(50);
    ProfileLaser 	: STRING(50);
END_STRUCT
END_TYPE

// ---- DUTs/Database/DUT_stBroachingPlan.TcDUT
TYPE DUT_stBroachingPlan :
STRUCT
    PassCount 		: DINT;
    Pass1BaseBroachingPlan 		: DUT_stBroachingPlanBase;
	Pass1VariantsBroachingPlan 	: DUT_stBroachingPlanVariants;
    Pass2BaseBroachingPlan 		: DUT_stBroachingPlanBase;
	Pass2VariantsBroachingPlan 	: DUT_stBroachingPlanVariants;
    Pass3BaseBroachingPlan 		: DUT_stBroachingPlanBase;
	Pass3VariantsBroachingPlan 	: DUT_stBroachingPlanVariants;
    Pass4BaseBroachingPlan 		: DUT_stBroachingPlanBase;
	Pass4VariantsBroachingPlan 	: DUT_stBroachingPlanVariants;
	Pass5BaseBroachingPlan 		: DUT_stBroachingPlanBase;
	Pass5VariantsBroachingPlan 	: DUT_stBroachingPlanVariants;
END_STRUCT
END_TYPE

// ---- DUTs/Database/DUT_stOrder.TcDUT
TYPE DUT_stOrder :
STRUCT
	Position				: DINT;
	BatchName				: STRING(50);
	Status					: STRING(50);
	ProductName				: STRING(50);
	BlankKeyType			: STRING(10);
	SideBar					: STRING(10);
	Quantity				: DINT;
	ExternMarkingData		: DUT_stExternMarkingData;
	Direct					: BOOL;
END_STRUCT
END_TYPE

// ---- DUTs/Database/DUT_stOrderItems.TcDUT
TYPE DUT_stOrderItems :
STRUCT
	return_			: DINT;
	BatchId	: STRING(50);
END_STRUCT
END_TYPE

// ---- DUTs/Database/DUT_stPLCData.TcDUT
TYPE DUT_stPLCData :
STRUCT
	PartId : DINT;
	RowIndex : STRING(50);
	RunningNo : STRING(50);
  	ProfileName : STRING(50);
  	FamilyName : STRING(50);
  	PlugType : STRING(50);
  	IsFirstPartInBatch : STRING(50);
  	IsLastPartInBatch : STRING(50);
  	IsFirstPartInRow : STRING(50);
  	IsLastPartInRow : STRING(50);
	MarkingData : DUT_stMarkingData;
	Brushing : STRING(50);
	BackHole : STRING(50);
	UnloadingModeId : DINT;
	BroachingPlan : DUT_stBroachingPlan;
END_STRUCT
END_TYPE

// ---- DUTs/Database/DUT_stProcessingData.TcDUT
TYPE DUT_stProcessingData :
STRUCT
	LocationId	: UINT;
	PartId		: LINT;
	StatusId	: eDbPiecesStatus;
	Status		: STRING(10);
	DefectId	: UINT;
	Defect		: STRING;
	ProcessingStartedAt	: STRING(39);
	ProcessingEndedAt	: STRING(39);
	IsInitialUpdate		: STRING(5);
	IsFinalUpdate		: STRING(5);
END_STRUCT
END_TYPE

// ---- DUTs/Database/DUT_stProcessingHMIData1.TcDUT
TYPE DUT_stProcessingHMIData1 :
STRUCT
	LocationId 			: DINT;
	PartId	 			: DINT;
END_STRUCT
END_TYPE

// ---- DUTs/Database/DUT_stProcessingHMIData2.TcDUT
TYPE DUT_stProcessingHMIData2 :
STRUCT
    ProductName 	: STRING(50);
	BatchName 		: STRING(50);
	RowIndex		: STRING(50);
	RowRunningNo    : STRING(50);
	RowQty          : STRING(50);
	OrderReference  : STRING(50);
	Profile         : STRING(50);
	PlugType		: STRING(50);
	Brushing        : STRING(50);
	ProfileLaser    : STRING(50);
	BackHole       	: STRING(50);
    UnloadMode 		: STRING(50);
    RunningNoOverRowQty : STRING(50);
	//CurrentRowOverRowCount  : STRING(50);
END_STRUCT
END_TYPE

// ---- DUTs/Database/DUT_stUpdateBatchToProductionQueue.TcDUT
TYPE DUT_stUpdateBatchToProductionQueue :
STRUCT
	return_			: DINT;
	BatchId	: STRING(DB.MAX_STRING_SIZE);
	BatchInfoJson	: STRING(DB.MAX_STRING_SIZE);
	BatchItemsJson	: STRING(DB.MAX_STRING_SIZE);
END_STRUCT
END_TYPE

// ---- DUTs/Database/DUT_UpdateCutterData.TcDUT
TYPE DUT_UpdateCutterData :
STRUCT
	Id		: DINT;
	Data	: STRING(DB.MAX_STRING_SIZE);
END_STRUCT
END_TYPE

// ---- DUTs/Database/DUT_UpdatePartLocationsAndProcessingData.TcDUT
TYPE DUT_UpdatePartLocationsAndProcessingData :
STRUCT
	return_value	: DINT;
	Data	: STRING(DB.MAX_STRING_SIZE);
END_STRUCT
END_TYPE

// ---- DUTs/Database/DUT_UpdateSettingRepositoryByName.TcDUT
TYPE DUT_UpdateSettingRepositoryByName:
STRUCT  
	return_value	: DINT;
	Name			: STRING(50);
	JsonValue		: STRING(DB.MAX_STRING_SIZE);
END_STRUCT
END_TYPE

// ---- DUTs/Database/eDbPiecesStatus.TcDUT
{attribute 'qualified_only'}
{attribute 'strict'}
TYPE eDbPiecesStatus :
(
	Scrap 		:= -1,
	Undefined	:= 0,
	Fetched		:= 1,
	Processing	:= 2,
	Completed	:= 3
);
END_TYPE

// ---- DUTs/Database/Mes/DUT_stMesOrder.TcDUT
TYPE DUT_stMesOrder :
STRUCT
	return_			: DINT;
	StatusFilter	: STRING(50);
	OrderListJson	: STRING(DB.MAX_STRING_SIZE);
END_STRUCT
END_TYPE

// ---- DUTs/Database/Mes/DUT_stMesOrderItems.TcDUT
TYPE DUT_stMesOrderItems :
STRUCT
	return_			: DINT;
	OrderReference	: STRING(50);
	OrderItemsJson	: STRING(DB.MAX_STRING_SIZE);
END_STRUCT
END_TYPE

// ---- DUTs/DUT_RobSetpoint_Real.TcDUT
TYPE DUT_RobSetpoint_Real :
STRUCT
	Override : USINT;
	PositionOffset : ARRAY[0..EC.NUM_ROBOT_OFFSET - 1] OF DUT_XYZ_Real;
END_STRUCT
END_TYPE

// ---- DUTs/DUT_XYZ_Real.TcDUT
TYPE DUT_XYZ_Real :
STRUCT
	X : REAL;
	Y : REAL;
	Z : REAL;
END_STRUCT
END_TYPE

// ---- DUTs/DUT_XYZ_Int.TcDUT
TYPE DUT_XYZ_Int :
STRUCT
	X : INT;
	Y : INT;
	Z : INT;
END_STRUCT
END_TYPE

// ---- DUTs/eDeviceType.TcTLEO
{attribute 'qualified_only'}
{attribute 'strict'}
TYPE eDeviceType :
(
	Unknown := 0,
	Primary := 1,
	Secondary := 2,
	Remote := 3
);
END_TYPE

// ---- DUTs/eLoadingMode.TcDUT
{attribute 'qualified_only'}
{attribute 'strict'}
TYPE eLoadingMode :
(
	Auto	  := 1,
	Manual	  := 2, 
	SemiAuto  := 3
);
END_TYPE

// ---- DUTs/DUT_Events.TcDUT
TYPE DUT_Events :
STRUCT
	wAlarm						: ARRAY[0..G.MAX_ALR_WORD] OF DWORD;						//Bit mask allarmi
	
	aAlarm						: ARRAY[0..G.MAX_ALR] OF FB_TcAlarm;
	
	Cumulative					: BOOL;
END_STRUCT
END_TYPE

// ---- DUTs/eBroach.TcDUT
{attribute 'qualified_only'}
{attribute 'strict'}
TYPE eBroach :
(
	Master	:= 0,
	V1		:= 2,
	V2		:= 3,
	V3		:= 4,
	V4		:= 5,
	V5		:= 6,
	V6		:= 7
);
END_TYPE

// ---- DUTs/DUT_DataRequest.TcDUT
TYPE DUT_DataRequest :
STRUCT
	aByte	: ARRAY[0..1] OF stByteAsBit; 	
	aDWord	: DWORD;
END_STRUCT
END_TYPE

// ---- DUTs/DUT_MachineData.TcDUT
TYPE DUT_MachineData :
STRUCT
	aBool	: ARRAY[0..79] OF BOOL; 	//10 byte -> 80 bool
	aByte	: ARRAY[0..10] OF USINT;	//10 byte -> 10 usint
	aWord	: ARRAY[0..14] OF UINT;		//60 byte -> 15 uint
	aSt	: ARRAY[1..19] OF DUT_StationData;
END_STRUCT
END_TYPE

// ---- DUTs/DUT_MATDiagnostics.TcDUT
TYPE DUT_MATDiagnostics :
STRUCT
    Running : BOOL;
    Heartbeat : BOOL;
    Error : BOOL;
    ErrorMessage : STRING(80);
END_STRUCT
END_TYPE

// ---- DUTs/DUT_St0Data.TcDUT
TYPE DUT_St0Data :
STRUCT
	FlagP	: ARRAY[0..5] OF BYTE; 	
	RunP	: DWORD;
	WindP	: DWORD;
	NpP		: DWORD;
	Tpcy	: BYTE;
	Tppz	: BYTE;
	TpcyS	: ARRAY[1..48] OF BYTE;
	Data	: ARRAY[1..93] OF DWORD;
	DataB	: ARRAY[1..20] OF BYTE;
	DataAu	: ARRAY[1..10] OF DWORD;
END_STRUCT
END_TYPE

// ---- DUTs/DUT_StationData.TcDUT
TYPE DUT_StationData :
STRUCT
	FlagP_B0 : BYTE;
	FlagP_B1 : BYTE;
	FlagP_B2 : BYTE;
	FlagP_B3 : BYTE;
	FlagP_B4 : BYTE;
	FlagP_B5 : BYTE;
	RunP_B0  : BYTE;
	RunP_B1  : BYTE;
	RunP_B2  : BYTE;
	RunP_B3  : BYTE;
	WidP_B0  : BYTE;
	WidP_B1  : BYTE;
	WidP_B2  : BYTE;
	WidP_B3  : BYTE;
	NppP_B0  : BYTE;
	NppP_B1  : BYTE;
	NppP_B2  : BYTE;
	NppP_B3  : BYTE;
	State    : BYTE;
	Byte_19  : BYTE;		
	Byte_20  : BYTE;		
	Byte_21  : BYTE;		
	Byte_22  : BYTE;		
	Byte_23  : BYTE;		
	Byte_24  : BYTE;		
	Byte_25  : BYTE;		
	Byte_26  : BYTE;		
	Byte_27  : BYTE;		
	Byte_28  : BYTE;		
	Byte_29  : BYTE;		
	Byte_30  : BYTE;		
	Byte_31  : BYTE;		
	Byte_32  : BYTE;		
	Byte_33  : BYTE;		
	Byte_34  : BYTE;		
	Byte_35  : BYTE;		
	Byte_36  : BYTE;		
	Byte_37  : BYTE;		
	Byte_38  : BYTE;		
	Byte_39  : BYTE;		
END_STRUCT
END_TYPE

// ---- DUTs/eConnectionSteps.TcDUT
TYPE eConnectionSteps :
(
	eCONNECTION_STATE_IDLE,
	eCONNECTION_STATE_CONNECT_START,
	eCONNECTION_STATE_CONNECT_WAIT,
	eCONNECTION_STATE_DATAEXCHANGE,
	eCONNECTION_STATE_CLOSE_START,
	eCONNECTION_STATE_CLOSE_WAIT,
	eCONNECTION_STATE_ERROR
);
END_TYPE

// ---- DUTs/eEV_Status.TcDUT
TYPE eEV_Status :
(
	NotUsed								:= -1,
	MovingForward						:= 0,
	MovingBackward						:= 1,
	MoveCompleted						:= 2,
	Timeout								:= 3,
	Error								:= 4
);
END_TYPE

// ---- DUTs/eHeaderPieces.TcTLEO
{attribute 'qualified_only'}
{attribute 'strict'}
TYPE eHeaderPieces :
(
	Ok 		:= 0,
	Ko 		:= 1,
	Loaded	:= 2,
	Total	:= 3,
	End		:= 4
);
END_TYPE

// ---- DUTs/eIcon.TcTLEO
{attribute 'qualified_only'}
{attribute 'strict'}
TYPE eIcon :
(
	Emg			:= 0,
	DoorOpen	:= 1,
	AirOk		:= 2,
	HydraulicOk	:= 3,
	EquipmentOk	:= 4,
	Home		:= 5,
	Connection	:= 6,
	End			:= 16
);
END_TYPE

// ---- DUTs/eMode.TcDUT
{attribute 'qualified_only'}
{attribute 'strict'}
TYPE eMode :
(
	MODE_MANUAL := 0,
	MODE_SINGLE := 1,
	MODE_AUTO := 2,
	MODE_MAINTENANCE := 3
);
END_TYPE

// ---- DUTs/eProductStatus.TcDUT
{attribute 'qualified_only'}
{attribute 'strict'}
TYPE eProductStatus :
(
	Scraped 	:= -1,
	NotPresent 	:= 0,
	Present 	:= 1,
	Working 	:= 2,
	Completed 	:= 3
);
END_TYPE

// ---- DUTs/eShiftPosMan.TcDUT
{attribute 'qualified_only'}
{attribute 'strict'}
TYPE eShiftPosMan :
(
	eSt0 := 0,
	eSt1 := 1,
	eSt2 := 2,
	eSt3 := 3,
	eSt4 := 4,
	eSt5 := 5,
	eSt6 := 6,
	eSt7 := 7,
	eSt8 := 8,
	eSt9 := 9,
	eSt10 := 10,
	eSt11 := 11,
	eSt12 := 12,
	eSt13 := 13,
	eSt14 := 14,
	eSt15 := 15,
	eSt16 := 16,
	eSt17 := 17,
	eSt18 := 18,
	eSt19 := 19,
	eSt20 := 20
);
END_TYPE

// ---- DUTs/eShiftPosPC100.TcDUT
{attribute 'qualified_only'}
{attribute 'strict'}
TYPE eShiftPosPC100 :
(
	eSt2b := 0,
	eSt2c := 1,
	eSt2d := 2
);
END_TYPE

// ---- DUTs/eState.TcTLEO
{attribute 'qualified_only'}
{attribute 'strict'}
TYPE eState :
(
	Undefine	:= -1,
	PowerOff	:= 0,
	Home		:= 1,
	Ready		:= 2,
	Running		:= 3,
	Alarm		:= 4,
	Emptying	:= 5,
	Loading		:= 6,
	Manual		:= 7,
	UpsOn		:= 99 //solo per database, creato internamente in PLC Beckhoff
);
END_TYPE
//  Undefine = '-1'

// ---- DUTs/eStationData.TcDUT
{attribute 'qualified_only'}
{attribute 'strict'}
TYPE eStationData :
(
	aSt1	:= 0,
	aSt2	:= 1,
	aSt3	:= 2,
	aSt4	:= 3,
	aSt5	:= 4,
	aSt6	:= 5,
	aSt7	:= 6,
	aSt8	:= 7,
	aSt9	:= 8,
	aSt10	:= 9,
	aSt11	:= 10,
	aSt12	:= 11,
	aSt13	:= 12,
	aSt14	:= 13,
	aSt15	:= 14,
	aSt16	:= 15,
	aSt2b	:= 16,
	aSt2c	:= 17,
	aSt2d	:= 18
);
END_TYPE

// ---- DUTs/eStationState.TcDUT
{attribute 'qualified_only'}
{attribute 'strict'}
TYPE eStationState :
(
	Alarm 		:= -1,
	Disable 	:= 0,
	Ready 		:= 1,
	Working		:= 2,
	EndOfJob	:= 3,
	Undefine	:= 4,
	Extraction	:= 5,
	Infeed		:= 6
);
END_TYPE

// ---- DUTs/EventsMgt/ST_EventClassInfo.TcDUT
TYPE ST_EventClassInfo :
STRUCT
	GUID : GUID;
	BaseAddress : POINTER TO TcEventEntry;
	Count : UDINT;
END_STRUCT
END_TYPE

// ---- DUTs/EventsMgt/ST_FanucCNCEventAxesMask.TcDUT
TYPE ST_FanucCNCEventAxesMask :
STRUCT
	Axis_1 : BIT;
	Axis_2 : BIT;
	Axis_3 : BIT;
	Axis_4 : BIT;
	Axis_5 : BIT;
	Axis_6 : BIT;
	Axis_7 : BIT;
	Axis_8 : BIT;
END_STRUCT
END_TYPE

// ---- DUTs/EventsMgt/ST_FanucCNCEventDetails.TcDUT
TYPE ST_FanucCNCEventDetails :
STRUCT
	AxesMask : ST_FanucCNCEventAxesMask;
	Category : BYTE;
	No : UINT;
END_STRUCT
END_TYPE

// ---- DUTs/EventsMgt/ST_FanucCNCEventEntryDetails.TcDUT
TYPE ST_FanucCNCEventEntryDetails :
STRUCT
	SourceInfo : U_FanucCNCEventSourceInfo;
	EventInfo : U_FanucCNCEventInfo;
END_STRUCT
END_TYPE

// ---- DUTs/EventsMgt/ST_FanucCNCEventSourceDetails.TcDUT
TYPE ST_FanucCNCEventSourceDetails :
STRUCT
	MainType : BYTE;
	SubType : BYTE;
	CNCNo : BYTE;
	PathNo : BYTE;
END_STRUCT
END_TYPE

// ---- DUTs/EventsMgt/ST_FanucCNCEventSourceInfo.TcDUT
TYPE ST_FanucCNCEventSourceInfo :
STRUCT
	SourceId : U_FanucCNCEventSourceInfo;		// 4 bytes					=  4
	CNCName : STRING[21];						// (21 + 1) bytes			= 22
	PathName : STRING[21];						// (21 + 1) bytes			= 22
	AxisNames : ARRAY [1..8] OF STRING[3];		// 8 * (3 + 1) = 32 bytes	= 32
END_STRUCT										//					Totale	= 80
END_TYPE

// ---- DUTs/EventsMgt/ST_FanucCNCEventSourceList.TcDUT
TYPE ST_FanucCNCEventSourceList :
STRUCT
	FanucCNCSources : ARRAY [1..NUM_MAX_CNC_EVENT_SOURCES] OF ST_FanucCNCEventSourceInfo;
	HashMD5 : ARRAY[0..15] OF BYTE;
END_STRUCT
END_TYPE

// ---- DUTs/EventsMgt/ST_FanucSourceDescriptor.TcDUT
TYPE ST_FanucSourceDescriptor :
STRUCT
	MainType : BYTE;
	SubType : BYTE;
	CNCNo : BYTE;
	PathNo : BYTE;
END_STRUCT
END_TYPE

// ---- DUTs/EventsMgt/U_FanucCNCEventEntry.TcDUT
TYPE U_FanucCNCEventEntry :
UNION
	{attribute 'displaymode':='hex'}
	Id : LWORD;
	Details : ST_FanucCNCEventEntryDetails;	
END_UNION
END_TYPE

// ---- DUTs/EventsMgt/U_FanucCNCEventInfo.TcDUT
TYPE U_FanucCNCEventInfo :
UNION
	{attribute 'displaymode':='hex'}
	Id : WORD;
	Details : ST_FanucCNCEventDetails;
END_UNION

END_TYPE

// ---- DUTs/EventsMgt/U_FanucCNCEventSourceInfo.TcDUT
TYPE U_FanucCNCEventSourceInfo :
UNION
	{attribute 'displaymode':='hex'}
	Id : DWORD;
	Details : ST_FanucCNCEventSourceDetails;
END_UNION

END_TYPE

// ---- DUTs/HMI/DUT_HIM_ProscessingData.TcDUT
TYPE DUT_HIM_ProscessingData :
STRUCT
	Name			: STRING(10);
	PartId			: DINT;
    ProductName 	: STRING(50);
	BatchName 		: STRING(50);
	RowIndex		: STRING(50);
	RowRunningNo    : STRING(50);
	RowQty          : STRING(50);
	OrderReference  : STRING(50);
	Profile 		: STRING(50);
	PlugType       	: STRING(50);
	Brushing     	: STRING(50);
	ProfileLaser    : STRING(50);
	BackHole        : STRING(50);
	UnloadMode      : STRING(50);
    RunningNoOverRowQty : STRING(50);
	CurrentRowOverRowCount  : STRING(50);	
	ProductStatus			: eProductStatus;
END_STRUCT
END_TYPE

// ---- DUTs/HMI/DUT_HIM_DeviceType.TcDUT
TYPE DUT_HIM_DeviceType :
STRUCT
	Ip : STRING(15);
	DeviceType : eDeviceType;
END_STRUCT
END_TYPE

// ---- DUTs/HMI/DUT_HMI_Display.TcDUT
TYPE DUT_HMI_Display :
STRUCT
	Enable: BOOL;
	Value:DINT;
END_STRUCT
END_TYPE

// ---- DUTs/HMI/DUT_HMI_Events.TcDUT
TYPE DUT_HMI_Events :
STRUCT
	Clear :BOOL;
END_STRUCT
END_TYPE

// ---- DUTs/HMI/DUT_HMI_EV_Diagnostic.TcDUT
TYPE DUT_HMI_EV_Diagnostic :
STRUCT
	Enable	 : BOOL;
	dFwdTime : UINT;
	dBwdTime : UINT;
	eStatus  : eEV_Status;
	Error 	 : BOOL;	
END_STRUCT
END_TYPE

// ---- DUTs/HMI/DUT_HMI_EV_Info.TcDUT
TYPE DUT_HMI_EV_Info :
STRUCT
	Enable	 : BOOL;
	dTime 	 : UINT;
	Error 	 : BOOL;	
END_STRUCT
END_TYPE

// ---- DUTs/HMI/DUT_HMI_General.TcDUT
TYPE DUT_HMI_General :
STRUCT
	Manuals 	: DUT_HMI_General_Manuals;		// Fanuc 
	Mes			: DUT_HMI_MesManual;
END_STRUCT
END_TYPE

// ---- DUTs/HMI/DUT_HMI_General_Manuals.TcDUT
TYPE DUT_HMI_General_Manuals :
STRUCT
	PS : ARRAY[0..CNC.NUM_MAX_MANUALS_GENERAL-1] OF BOOL;
	LS : ARRAY[0..CNC.NUM_MAX_MANUALS_GENERAL-1] OF BOOL;
END_STRUCT
END_TYPE

// ---- DUTs/HMI/DUT_HMI_Header.TcDUT
TYPE DUT_HMI_Header :
STRUCT
	OperatingMode	: eMode;
	MachineState	: eState;
	Override 		: STRING(3);
	OvrMultiplier	: STRING(3);
	OvrMultFeedback	: BOOL;
	Feedrate 		: STRING(3);
	Icons			: ARRAY[0..eIcon.End] OF BOOL;
	Equipment 		: STRING;
	Pieces			: ARRAY[0..eHeaderPieces.End] OF UDINT;
	ProgressBar		: USINT;
	PathActive		: STRING(2);
END_STRUCT
END_TYPE

// ---- DUTs/HMI/DUT_HMI_In.TcDUT
TYPE DUT_HMI_In :
STRUCT
	AxisSelected 		: USINT;
	Tools				: DUT_HMI_Tools;
	Header				: DUT_HMI_Header;
	Events				: DUT_HMI_Events;
	Navigation			: DUT_HMI_Navigation;
	Dummy				: ARRAY[0..9] OF BOOL; // Non ho capito perchè ma in qualche modo pannelo scrive più memoria oltre in navigation, quindi ho dichiarato questa variabile
												// per occupare memoria a caso, se no pannello mi tenva forzata la roba di statistics
	Statistics			: DUT_Statistics;
	Resource			: DUT_HMI_In_Resource;
	LoadingModeChanged  : BOOL;
END_STRUCT
END_TYPE

// ---- DUTs/HMI/DUT_HMI_In_Resource.TcDUT
TYPE DUT_HMI_In_Resource :
STRUCT
	ProductName		: STRING(50);
	Refresh			: BOOL;
END_STRUCT
END_TYPE

// ---- DUTs/HMI/DUT_HMI_MesManual.TcDUT
TYPE DUT_HMI_MesManual :
STRUCT
	PS : BOOL;
	LS : BOOL;
	Data : STRING(DB.MAX_STRING_SIZE);
END_STRUCT
END_TYPE

// ---- DUTs/HMI/DUT_HMI_Navigation.TcDUT
TYPE DUT_HMI_Navigation :
STRUCT
	PS : ARRAY[0..HMI.NUM_NAVIGATION_ITEMS-1] OF BOOL;
	LS : ARRAY[0..HMI.NUM_NAVIGATION_ITEMS-1] OF BOOL;
END_STRUCT
END_TYPE

// ---- DUTs/HMI/DUT_HIM_Probe.TcDUT
TYPE DUT_HIM_Probe :
STRUCT
	ActualProbeValue : REAL;
	ActualEncoderValue : REAL;
	Error	: BOOL;
	UpperLimit	: REAL;
	LowerLimit	: REAL;
END_STRUCT
END_TYPE

// ---- DUTs/HMI/DUT_HMI_Out.TcDUT
TYPE DUT_HMI_Out :
STRUCT
	UPSDiagnostic 	: DUT_HMI_UPSStatus;
	Header		  	: DUT_HMI_Header;
	AxisSelected  	: USINT;
	Tools			: DUT_HMI_Tools;
	OrderList 		: ARRAY[0..G.PRODUCTIONTABLE_SIZE] OF DUT_stOrder;
	Doors			: ARRAY[0..5] OF SINT;
	Gc1000Status	: SINT;
	Resource		: DUT_HMI_Out_Resource;
	Probe			: DUT_HIM_Probe;
	CycleTime		: STRING(50);
	Counters		: DUT_HMI_Production_Counters;
	ProductionQueueRefresh : BOOL;
	KebaEnabled	: BOOL;
	KebaHMILoaded : BOOL;
	IpDevices	: ARRAY[0..1] OF DUT_HIM_DeviceType;
	EnableProductionAction: BOOL;
	ResfreshPermissions : BOOL;
END_STRUCT
END_TYPE

// ---- DUTs/HMI/DUT_HMI_Out_Resource.TcDUT
TYPE DUT_HMI_Out_Resource :
STRUCT
	Origin : DUT_OutInfoOrigin;
END_STRUCT
END_TYPE

// ---- DUTs/HMI/DUT_HMI_Production_Counters.TcDUT
TYPE DUT_HMI_Production_Counters :
STRUCT
	TotalPieceGood : UDINT;
	TotalPieceScrap : UDINT;
END_STRUCT
END_TYPE

// ---- DUTs/HMI/DUT_HMI_Tools.TcDUT
TYPE DUT_HMI_Tools :
STRUCT
	TaskManager			: BOOL; // Open Windows Task Manager program
	CNCScreenDisplay 	: BOOL; // Open Fancu CNC Screen Display program
	ProgramTransferTool : BOOL; // Open Fanuc Program Transfer Tool program
	OnScreenKeyboard	: BOOL; // Open On Screen Kryboard tool
	CloseBrowser		: BOOL; // Close browser and HMI application
	FanucLadder			: BOOL; // Open Fanuc Ladder program
	FlyCad				: BOOL; // Open Lasit FlyCad software
	OpenPage			: BOOL; // Open tools page
END_STRUCT
END_TYPE

// ---- DUTs/HMI/DUT_HMI_UPSStatus.TcDUT
TYPE DUT_HMI_UPSStatus :
STRUCT
	Valid : BOOL;
	State : ST_UPSStatus;
END_STRUCT
END_TYPE

// ---- DUTs/Production/DUT_Production.TcDUT
TYPE DUT_Production :
STRUCT
	Counters				: DUT_Production_Counters; // Piece Counters
	OEE						: DUT_Production_OEE; // OEE Parameters
END_STRUCT
END_TYPE

// ---- DUTs/Production/DUT_Production_Counters.TcDUT
TYPE DUT_Production_Counters :
STRUCT
	TotalPieces						: UDINT; 	// Contatore totale pezzi
	PartialPieces					: UDINT; 	// Contatore pezzi resettabile manualmente
	PartialActualGood				: UDINT;	// COntatore pezzi buoni resettabile manualmente
	BatchPieces						: UDINT;	// Pezzi da produrre per il lotto
	ActualGood						: UDINT;	// Pezzi ok
	ActualPieces					: DINT;		// Pezzi già prodotti per il lotto
	ActualScrap						: DINT;		// Pezzi già prodotti per il lotto
	PiecesPerHour 					: ARRAY[0..23] OF REAL;
	MaxPiecesPerHour 				: REAL;
	ActualDate						: ARRAY [0..2] OF WORD;
	ActivePiecesDaily_PreviousHours	: REAL;
	Pieces_Daily					: REAL;
	BatchPiecesUpdateConfirm		: BOOL;
	BatchPiecesUpdateAbort			: BOOL;
	BatchPiecesTextInputValue		: UDINT;
END_STRUCT
END_TYPE

// ---- DUTs/Production/DUT_Production_OEE.TcDUT
TYPE DUT_Production_OEE :
STRUCT
	Availabilty 			: REAL;
	Performance 			: REAL;
	Quality					: REAL;
	tON						: REAL; // Tempo di reale produzione in Production Mode
	tOFF					: REAL; // Tempo di attesa operatore in Production Mode
	tDOWN					: REAL; // Tempo di macchina in uno stato che non può produrre
	s_tON					: STRING; // Tempo di reale produzione in Production Mode
	s_tOFF					: STRING; // Tempo di attesa operatore in Production Mode
	s_tDOWN					: STRING; // Tempo di macchina in uno stato che non può produrre
	s_tTOTAL				: STRING; // Tempo di osservazione
	OEE						: REAL;
	GoodPieces				: DINT;
	BadPieces				: DINT;
	IdealCycleTime			: TIME := T#9s;
	PlannedProductionTime	: DWORD := 60;
	OperatingTime			: TIME;
END_STRUCT
END_TYPE

// ---- DUTs/Production/DUT_Statistics.TcDUT
TYPE DUT_Statistics :
STRUCT
	OEE_Enable				: BOOL;
	OEE_Reset				: BOOL;
END_STRUCT
END_TYPE

// ---- DUTs/Production/eOEE.TcDUT
{attribute 'qualified_only'}
{attribute 'strict'}
TYPE eOEE :
(
	Downtime 	:= 0,
	Uptime	 	:= 1,
	Pause		:= 2,
	Completed	:= 3
);
END_TYPE

// ---- DUTs/stBit.TcDUT
TYPE stBit :
STRUCT
    b0  : BIT;
    b1  : BIT;
    b2  : BIT;
    b3  : BIT;
    b4  : BIT;
    b5  : BIT;
    b6  : BIT;
    b7  : BIT; 
END_STRUCT
END_TYPE

// ---- DUTs/stByteAsBit.TcDUT
TYPE stByteAsBit :
UNION
	aByte	: BYTE;
	aBit	: stBit;
END_UNION
END_TYPE

// ---- DUTs/stTestStringUnion.TcDUT
TYPE stTestStringUnion :
UNION
	sString		: STRING(DB.MAX_STRING_SIZE);
	nByte		: ARRAY[0..DB.MAX_STRING_SIZE] OF BYTE;
END_UNION
END_TYPE

// ---- DUTs/stFanucCNCKeyboard.TcDUT
TYPE stFanucCNCKeyboard :
STRUCT
	PS: ARRAY[0..(NUM_MAX_CNC_KEYBOARD_FOR_BECKHOFF-1)] OF BOOL;
	LS: ARRAY[0..(NUM_MAX_CNC_KEYBOARD_FOR_BECKHOFF-1)] OF BOOL;
END_STRUCT
END_TYPE

// ---- DUTs/stShiftData.TcDUT
TYPE stShiftData :
STRUCT
	FLAGP : stByteAsBit;
	WIDP : DINT;
	
	PmcData : DUT_St0Data;
	stPLCData 			: DUT_stPLCData;
	ProcessingData 		: DUT_stProcessingHMIData2;
END_STRUCT
END_TYPE

// ---- DUTs/DataBuffer.TcDUT
TYPE DataBuffer :
STRUCT
	WIDP : DINT;
	PmcData : DUT_St0Data;
	stPLCData 			: DUT_stPLCData;
END_STRUCT
END_TYPE

// ---- FBs/LaserMarker - LASIT/DUT_Job.TcDUT
TYPE DUT_Job :
STRUCT
	JobName			: STRING(50);
	JobIndex		: USINT;
	IndexDynamicCmd	: ARRAY[1..10] OF BOOL;
END_STRUCT
END_TYPE

// ---- GVLs/CNC.TcGVL
VAR_GLOBAL CONSTANT
// Events
	NUM_CNC_EVENTS 					: UINT := 5000;	
	NUM_PMC_EVENTS 					: UINT := 4000;
	NUM_MAX_CNC_ACTIVE_EVENTS 		: UINT := 50;
	NUM_MAX_CNC_EVENT_SOURCES 		: UINT := 50;
	NUM_MAX_STATION_ALARMS			: UINT := 80;
	NUM_MAX_STATION_WARNINGS		: UINT := 16;
	NUM_MAX_GENERAL_ALARMS			: UINT := 160;
	NUM_MAX_GENERAL_WARNINGS		: UINT := 200;
	NUM_00_ALARMS					: UINT := 300;
	NUM_00_WARNINGS					: UINT := 100;
	
// Navigation
	NUM_NAVIGATION_ITEMS 			: UINT := 3;	// Numero di byte scritti su pmc
	
// Keyboard layout	
	NUM_MAX_CNC_KEYBOARD_FOR_BECKHOFF 	: UINT := 64;
	NUM_MAX_CNC_KEYBOARD			: UINT := 8;

// Buttons and leds	
	NUM_MAX_CNC_BUTTONS_LEDS  		: UINT := 500;
	
// HS
	NUM_HS_EACH_STATION				: UINT := 50;
	
// Number of stations
	NUM_STATIONS					: UINT := 9;
	NUM_DATA_POSITION				: UINT := 14;
	
	NUM_MAX_MANUALS_GENERAL 		: UINT := 480;
	NUM_MAX_MANUALS_00 				: UINT := 320;
	NUM_MAX_MANUALS_01 				: UINT := 80;
	NUM_MAX_MANUALS_02 				: UINT := 80;
	NUM_MAX_MANUALS_03 				: UINT := 80;
	NUM_MAX_MANUALS_04 				: UINT := 80;
	NUM_MAX_MANUALS_05 				: UINT := 80;
	NUM_MAX_MANUALS_06 				: UINT := 80;
	NUM_MAX_MANUALS_07 				: UINT := 80;
	NUM_MAX_MANUALS_08 				: UINT := 80;
	NUM_MAX_MANUALS_09 				: UINT := 80;
	NUM_MAX_MANUALS_10 				: UINT := 80;
	NUM_MAX_MANUALS_11 				: UINT := 80;
	NUM_MAX_MANUALS_12 				: UINT := 80;
	NUM_MAX_MANUALS_13 				: UINT := 80;
	NUM_MAX_MANUALS_14 				: UINT := 80;
	NUM_MAX_MANUALS_15 				: UINT := 80;
	NUM_MAX_MANUALS_16 				: UINT := 80;
	NUM_MAX_MANUALS_17 				: UINT := 80;
	NUM_MAX_MANUALS_18 				: UINT := 80;
	
	IPAddress						: STRING := '192.168.1.1';
END_VAR

{attribute 'qualified_only'}
VAR_GLOBAL
	vKeyboard : stFanucCNCKeyboard;
	MachineData	: DUT_MachineData;
	MachineStatus : ARRAY[1..4] OF USINT;
	DataRequestRead : DUT_DataRequest;
	DataRequestWrite : DUT_DataRequest;
	
// MAT - Data exchange FOCAS-ADS
// vKeyboard	
	Q_R3900 AT %MB3000 	: ARRAY[0..(NUM_MAX_CNC_KEYBOARD-1)] OF BYTE; // vKeyboard - Keys Area 
	MATDiagnostic_MB3000 : DUT_MATDiagnostics;
	I_R3950 AT %MB3500 	: ARRAY[0..(NUM_MAX_CNC_KEYBOARD-1)] OF BYTE; // vKeyboard - Leds Area 
	MATDiagnostic_MB3500 : DUT_MATDiagnostics;
	
// Buttons/Leds
	Q_R4000 AT %MB14000 : ARRAY[0..(NUM_MAX_CNC_BUTTONS_LEDS-1)] OF BYTE; // Buttons
	MATDiagnostic_MB14000 : DUT_MATDiagnostics;
	I_R4500 AT %MB14500 : ARRAY[0..(NUM_MAX_CNC_BUTTONS_LEDS-1)] OF BYTE; // Leds
	MATDiagnostic_MB14500 : DUT_MATDiagnostics;
			
// MachineData
	I_E0000 AT %MB8000 : ARRAY[0..1999] OF BYTE;
	MATDiagnostic_MB8000 : DUT_MATDiagnostics;
	
// St0 Data
	St0Data AT %MB20000 : ARRAY[0..499] OF BYTE;
	St0DataTemp : DUT_St0Data;
	MATDiagnostic_MB20000 : DUT_MATDiagnostics;
	
// HS_write
	HS_write AT %MB4000 : ARRAY[0..12] OF BYTE;
	MATDiagnostic_MB4000 : DUT_MATDiagnostics;	

// HS_read
	HS_read AT %MB6000 : ARRAY[0..9] OF BYTE;
	MATDiagnostic_MB6000 : DUT_MATDiagnostics;
	
// FlyPowerOn // scritto da MatManager
	FlyPowerMarkOn	: BYTE;
	
// ProfiNET
	Q_X400 	AT %Q* : ARRAY[0..99] OF BYTE; // ProfiNET - To CNC
	Q_R2000 AT %Q* : ARRAY[0..199] OF BYTE; // ProfiNET - To CNC
	Q_D2000 AT %Q* : ARRAY[0..199] OF BYTE; // ProfiNET - To CNC
	
	I_Y400 	AT %I* : ARRAY[0..99] OF BYTE; // ProfiNET - From CNC
	I_R2200 AT %I* : ARRAY[0..199] OF BYTE; // ProfiNET - From CNC
	I_D2200 AT %I* : ARRAY[0..199] OF BYTE; // ProfiNET - From CNC
END_VAR

// ---- GVLs/DB.TcGVL
{attribute 'qualified_only'}
VAR_GLOBAL CONSTANT
	PRODUCTION_QUEUE_BUFFER_DIM : UINT := 50;
	MAX_STRING_SIZE	: UDINT := 65535;
	MAX_NUMBER_ST	: UDINT := 79;
END_VAR

VAR_GLOBAL
	stPLCData 			: DUT_stPLCData;
	stOrder 			: ARRAY[0..DB.PRODUCTION_QUEUE_BUFFER_DIM] OF DUT_stOrder;
	stProcessingData	: ARRAY[0..CNC.NUM_STATIONS] OF DUT_stProcessingData;
	
	ProcessingHMIDataLocation	: ARRAY[0..CNC.NUM_DATA_POSITION] OF DUT_stProcessingHMIData1;
	ProcessingHMIDataViewData	: ARRAY[0..CNC.NUM_DATA_POSITION] OF DUT_stProcessingHMIData2;
	
	stResourceInfo			: ARRAY[0..6] OF DUT_OutInfoOrigin;
	fbTriggerSequencer 		: FB_TriggerSequencer;
	
	HMI_SP_Alarm			: ARRAY[1..DB.MAX_NUMBER_ST] OF DUT_stSPAlarm;
	MesReadStatusCmd	: BOOL;
	GetProcessingDataForHMI_Trig : BOOL;
	
/////////////FOR HMI
	fbGSCNextSPGetResourcesByType : FB_MSSQL_spGetResourcesByType; // usato direttemente da HMI
	fbGSCNextSPGetResourcesByName : FB_MSSQL_spGetResourcesByName; // usato direttemente da HMI
	fbGSCNextSPSetResourcesByName : FB_MSSQL_spSetResourcesByName; // usato direttemente da HMI
	fbGSCNextSPGetResourcesListByType : FB_MSSQL_spGetResourcesListByType; // usato direttemente da HMI
	fbGSCNextSPGetFormattedTablesFromSequences : FB_MSSQL_spGetFormattedTablesFromSequences; // usato direttemente da HMI
	fbGSCNextSPGetOriginsFromSequence 	: FB_MSSQL_spGetOriginsFromSequence; // usato direttemente da HMI
	fbGSCNextSPGetBlankKey 				: FB_MSSQL_spGetBlankKey; // usato direttemente da HMI
	fbGSCNextSPGetBlankKeyByName 		: FB_MSSQL_spGetBlankKeyByName; // usato direttemente da HMI
	fbGSCNextSPGetBatchHistory   		: FB_MSSQL_spGetBatchHistory; // usato direttemente da HMI
	fbGSCNextSPGetBatchHistoryByStatus 	: FB_MSSQL_spGetBatchHistoryByStatus; // usato direttemente da HMI
	fbGSCNextSPGetPartHistory  			: FB_MSSQL_spGetPartHistory; // usato direttemente da HMI
	fbGSCNextSPGetPartHistoryByBatchName : FB_MSSQL_spGetPartHistoryByBatchName; // usato direttemente da HMI
	fbGSCNextSPGetSideCode 				: FB_MSSQL_spGetSideCode; // usato direttemente da HMI
	fbGSCNextSPGetOrigins 				: FB_MSSQL_spGetOrigins; // usato direttemente da HMI
	fbGSCNextSPGetOriginsByName 		: FB_MSSQL_spGetOriginsByName; // usato direttemente da HMI
	fbGSCNextSPGetOriginsBySide 		: FB_MSSQL_spGetOriginsBySide; // usato direttemente da HMI
	fbGSCNextSPGetCutters 				: FB_MSSQL_spGetCutters; // usato direttemente da HMI
	fbGSCNextSPGetCuttersByName			: FB_MSSQL_spGetCuttersByName; // usato direttemente da HMI
	fbGSCNextSPGetCuttersBySide 		: FB_MSSQL_spGetCuttersBySide; // usato direttemente da HMI
	fbGSCNextSPGetMillings 				: FB_MSSQL_spGetMillings; // usato direttemente da HMI
	fbGSCNextSPGetMillingsByName 		: FB_MSSQL_spGetMillingsByName; // usato direttemente da HMI
	fbGSCNextSPGetMillingsByFamilyName 	: FB_MSSQL_spGetMillingsByFamilyName; // usato direttemente da HMI
	fbGSCNextSPGetResourcesByNameMilling 	: FB_MSSQL_spGetResourcesByNameMilling; // usato direttemente da HMI
	fbGSCNextSPGetOrderInfoList 			: FB_MSSQL_spGetOrderInfoList; // usato direttemente da HMI
	fbGSCNextSPMES_GetOrderInfoList 		: FB_MSSQL_spMES_GetOrderInfoList; // usato direttemente da HMI
	fbGSCNextSPAppendBatchToProductionQueue : FB_MSSQL_spAppendBatchToProductionQueueFromHMI; // usato direttemente da HMI
	fbGSCNextSPMES_GetOrderItems 			: FB_MSSQL_spMES_GetOrderItems; // usato direttemente da HMI
	fbGSCNextSPGetOrderItems 			: FB_MSSQL_spGetOrderItems; // usato direttemente da HMI
	fbGSCNextSPGetBatchList				: ARRAY[0..1] OF FB_MSSQL_spGetBatchList; // usato direttemente da HMI
	fbGSCNextSPUpdateBatchToProductionQueue : FB_MSSQL_spUpdateBatchToProductionQueue; // usato direttemente da HMI
	fbGSCNextSPDeleteBatchToProductionQueue : FB_MSSQL_spDeleteBatchToProductionQueue; // usato direttemente da HMI
	fbGSCNextSPGetBatchHistoryDetail : FB_MSSQL_spGetBatchHistoryDetail; // usato direttemente da HMI
	fbGSCNextSPCMD_ForceCompletedBatch 	: FB_MSSQL_spCMD_ForceCompletedBatch; // usato direttemente da HMI
	fbGSCNextSPCMD_HoldBatch 			: FB_MSSQL_spCMD_HoldBatch; // usato direttemente da HMI
	fbGSCNextSPCMD_RecoverBatch 		: FB_MSSQL_spCMD_RecoverBatch; // usato direttemente da HMI
	fbGSCNextSPCMD_RestartBatch 		: FB_MSSQL_spCMD_RestartBatch; // usato direttemente da HMI
	fbGSCNextSPCMD_ResumeBatch 			: FB_MSSQL_spCMD_ResumeBatch; // usato direttemente da HMI
	fbGSCNextSPCMD_SuspendBatch 		: FB_MSSQL_spCMD_SuspendBatch; // usato direttemente da HMI
	fbGSCNextSPCMD_UnholdBatch 			: FB_MSSQL_spCMD_UnholdBatch; // usato direttemente da HMI
	fbGSCNextSPUpdateSettingRepositoryByName : FB_MSSQL_spUpdateSettingRepositoryByName;  // usato direttemente da HMI
	fbGSCNextSPGetSettingRepositoryList : FB_MSSQL_spGetSettingRepositoryList;  // usato direttemente da HMI	
	fbGSCNextSPGetBatchDetailById		: FB_MSSQL_spGetBatchDetailById;  // usato direttemente da HMI
	fbGSCNextSPChangeBatchPositionInProductionQueue: FB_MSSQL_spChangeBatchPositionInProductionQueue; // usato direttemente da HMI
	fbGSCNextSPGetCuttersOnDrum				: FB_MSSQL_spGetCuttersOnDrum; // usato direttemente da HMI
	fbGSCNextSPGetCuttersComboboxFormatted 	: FB_MSSQL_spGetCuttersComboboxFormatted; // usato direttemente da HMI
	fbGSCNextSPUpdateCuttersOnDrum 			: FB_MSSQL_spUpdateCuttersOnDrum; // usato direttemente da HMI
	fbGSCNextSPCheckCutterAlreadyPresentOnDrums: FB_MSSQL_spCheckCutterAlreadyPresentOnDrums; // usato direttemente da HMI
	fbGSCNextSPUpdateCutterData 			: FB_MSSQL_spUpdateCutterData; // usato direttemente da HMI
	fbGSCNextSPGetProfilesByFamilyName		: FB_MSSQL_spGetProfilesByFamilyName; // usato direttemente da HMI
	fbGSCNextSPGetProfiles 					: FB_MSSQL_spGetProfiles; // usato direttemente da HMI
	fbGSCNextSPGetFamilyNamesForCombobox	: FB_MSSQL_spGetFamilyNamesForCombobox; // usato direttemente da HMI
	fbGSCNextSPGetCuttersFromFamilyName		: FB_MSSQL_spGetCuttersFromFamilyName; // usato direttemente da HMI
	fbGSCNextSPDeleteProfile 				: FB_MSSQL_spDeleteProfile; // usato direttemente da HMI
	fbGSCNextSPAddProfile	 				: FB_MSSQL_spAddProfile; // usato direttemente da HMI
	fbGSCNextSPDeleteCutter 				: FB_MSSQL_spDeleteCutter; // usato direttemente da HMI
	fbGSCNextSPAddCutter 					: FB_MSSQL_spAddCutter; // usato direttemente da HMI
	fbGSCNextSPGetBroachingProfileSettings 	: FB_MSSQL_spGetBroachingProfileSettings; // usato direttemente da HMI
	fbGSCNextSPUpdateBroachingProfileSettings 	: FB_MSSQL_spUpdateBroachingProfileSettings; // usato direttemente da HMI
	fbGSCNextSPGetSettingRepositoryByName	: FB_MSSQL_spGetSettingRepositoryByName;  // usato direttemente da HMI
END_VAR

// ---- GVLs/EC.TcGVL
VAR_GLOBAL CONSTANT
	sNetId : STRING := '192.168.2.200.1.1';
	NUM_ROBOT_OFFSET : UINT := 4;
	NUM_MAX_ROBOT_OVR : UINT := 100;
	NUM_MAX_BROACH : UINT := 24;
	NUM_MIN_BROACH : UINT := 1;
END_VAR

VAR_GLOBAL
	EtherCAT_DevState AT %I* : UINT;
	ProfiNET_DevState AT %I* : UINT;

// FESTO	
	AL671 AT %Q* : ARRAY[0..4] OF UINT; // EV1-EV27
	AL673 AT %Q* : ARRAY[0..5] OF UINT; // EV28-EV55
	
// Override 
	I_Ovr_CounterValue 		AT %I* : UINT;
	I_Ovr_SetCounterDone 	AT %I* : BOOL;
	
	Q_Ovr_SetCounter 		AT %Q* : BOOL;
	Q_Ovr_SetCounterValue 	AT %Q* : UINT;
	
	I_Ovr_Overflow			AT %I* : BOOL;
	I_Ovr_Underflow			AT %I* : BOOL;
END_VAR

// ---- GVLs/ETH.TcGVL
VAR_GLOBAL CONSTANT
	PLCPRJ_BUFFER_SIZE						: UDINT := 1000;

	PLCPRJ_RECEIVE_POLLING_TIME		 		: TIME := T#10MS;
	PLCPRJ_RECEIVE_TIMEOUT					: TIME := T#10S;

	(* Some project specific error codes *)
	PLCPRJ_ERROR_RECEIVE_TIMEOUT			: UDINT := 16#8101;(* Receive timeout error *)
	PLCPRJ_ERROR_SENDFIFO_OVERFLOW			: UDINT := 16#8102;(* Send fifo overflow *)
	PLCPRJ_ERROR_RECFIFO_OVERFLOW			: UDINT := 16#8103;(* Receive fifo overflow *)
	UTF8_BOM								: STRING := 'ï»¿';
	END_LINE								: STRING := '$0D$0A';
	END_LINE_ANSWER							: STRING := '$R$N';
	
	SOH										: STRING := '$01';
	STX										: STRING := '$02';
	ETX										: STRING := '$03';
	EOT										: STRING := '$04';
	ACK										: STRING := '$06';
	ESC										: STRING := '$27';
END_VAR

// ---- GVLs/G.TcGVL
{attribute 'qualified_only'}
VAR_GLOBAL PERSISTENT RETAIN
	Ovr_CounterValue : UINT;
	Ovr : USINT;
	//ShiftManData : ARRAY[0..20] OF stShiftData;
	DataBuffer : ARRAY[0..DATABUFFER_SIZE] OF DataBuffer;
	filesList	: ARRAY[0..99] OF STRING;	
	filesNumb : UINT;   

	WID_Old : DINT;  
	Batch_old	:STRING; 

	LoadingModeActive : eLoadingMode;  
	OperatingModeOld : eMode;
	MachineStateOld	: eState;         
	IdList_Old	: ARRAY[0..10] OF DINT;
END_VAR
VAR_GLOBAL
	fbGetCurTaskIndex : GETCURTASKINDEX;
	
	RequestNext			: BOOL;
	RequestActual		: BOOL;
	
	SystemTime			: DT;
	
	ResetButton		: BOOL;
	MachineEmpty		: BOOL;
	
	fbProcessingData			: ARRAY[0..CNC.NUM_DATA_POSITION] OF FB_ProcessingData;
	
	PMCShiftDataSlide		: stShiftData;
	PMCShiftDataLaser		: stShiftData;
	PMCShiftDataCart		: stShiftData;
	PMCShiftDataDeburring	: stShiftData;
	PMCShiftDataPallet		: stShiftData;


	OEE_bCountUpGood  : BOOL;
	OEE_bCountUpBad  : BOOL;

	LasitOn				: BOOL;
	UpdatePartLocationsAndProcessingDataTrigger : BOOL;
END_VAR
VAR_GLOBAL CONSTANT
	PRODUCTIONTABLE_SIZE		: UDINT := 50;
	DATABUFFER_SIZE		: UINT := 50;
	MAX_ALR						: UINT 	:= 600;
	MAX_ALR_WORD				: UINT 	:= 60;
END_VAR

// ---- GVLs/HMI.TcGVL
{attribute 'qualified_only'}
VAR_GLOBAL CONSTANT
	NUM_NAVIGATION_ITEMS : UINT := 22;
END_VAR

VAR_GLOBAL PERSISTENT RETAIN
// Shifting Data from CNC
	ShiftData 	: ARRAY[0..20] OF stShiftData;
	Production		: DUT_Production;
	
	ContadinoBool	: BOOL;
	ContadinoString	: STRING;
	ProductsLoaded	: ARRAY[0..1] OF STRING;
	ProcessingData	: ARRAY[0..CNC.NUM_DATA_POSITION] OF DUT_HIM_ProscessingData;
	SelectedLoadingMode : eLoadingMode;
	ChipConveyorSetpoint	: UINT;
	DropsaSetpoint	: UINT;
	RobotLoadSetpoint : DUT_RobSetpoint_Real;
	RobotUnloadSetpoint : DUT_RobSetpoint_Real;
END_VAR

VAR_GLOBAL
	General		: DUT_HMI_General; 
	St0			: DUT_HMI_00;
	St1			: DUT_HMI_01;
	St2			: DUT_HMI_02;
	St3			: DUT_HMI_03;
	St4			: DUT_HMI_04;
	St5			: DUT_HMI_05;
	St6			: DUT_HMI_06;
	St7			: DUT_HMI_07;
	St8			: DUT_HMI_08;
	St9			: DUT_HMI_09;
	St10		: DUT_HMI_10;
	St11		: DUT_HMI_11;
	St12		: DUT_HMI_12;
	St13		: DUT_HMI_13;
	St14		: DUT_HMI_13;
	
//Shift Data
	ShiftTrigger : BOOL;
	ShiftnDone	 : BOOL;
	ShiftError	 : BOOL;	
	
// HMI Exchange	
	In  : DUT_HMI_In;
	Out : DUT_HMI_Out;
		
END_VAR

// ---- FBs/Events/I_EventDetailer.TcIO
INTERFACE I_EventDetailer

METHOD GetDetail : STRING(255)
VAR_INPUT
	TcAlarm : REFERENCE TO FB_TcAlarm;
END_VAR
END_METHOD

END_INTERFACE

// ---- FBs/StringBuilder/I_LimitedStringBuilder.TcIO
INTERFACE I_LimitedStringBuilder

METHOD  Append : I_StringBuilder // Append text to t current build string.
VAR_INPUT
	Text : STRING; //Text to append to current build string
END_VAR
END_METHOD

METHOD Left : I_StringBuilder
VAR_INPUT
	Count : INT;
END_VAR
END_METHOD

PROPERTY Length : INT
GET
END_GET
END_PROPERTY

METHOD Reset : I_LimitedStringBuilder //Reset current build string to an empty string.
END_METHOD

METHOD Right : I_StringBuilder
VAR_INPUT
	Count : INT;
END_VAR
END_METHOD

METHOD ToString : STRING //Returns current build string.
END_METHOD

END_INTERFACE

// ---- FBs/StringBuilder/I_StringBuilder.TcIO
INTERFACE I_StringBuilder

METHOD  Append : I_StringBuilder // Append text to t current build string.
VAR_INPUT
	Text : STRING; //Text to append to current build string
END_VAR
END_METHOD

METHOD InsertAtLocation : I_StringBuilder
VAR_INPUT
	Text : STRING;
	Position : INT;
END_VAR
END_METHOD

METHOD Reset : I_LimitedStringBuilder //Reset current build string to an empty string.
END_METHOD

METHOD ToString : STRING //Returns current build string.
END_METHOD

END_INTERFACE

// ---- POUs/MAIN.TcPOU
PROGRAM MAIN
VAR
	i					: UINT;
	ii					: UINT;
	fbGetCurTaskIndex 	: GETCURTASKINDEX;
	_iDataPos 			: INT;
	_dDataOff 			: DINT;	
	
	LasitManager : FB_LasitManager;
	Lasit 		: FB_Lasit;
	LasitFlyPowerMarkManager : FB_FlyPowerMarkManager;
	St04_MarkingData : DUT_stMarkingData;
	
	fbFlyPowerMarkExeManager : FB_FlyPowerMarkExeManager;
	fbFlyPowerMarkExeManagerInit : BOOL;

// ShiftData	
	stTempData  		: stShiftData;
	//fbShiftManData 		: FB_PartDataManager;
	fbShiftDataBuffer 	: FB_DataBufferManager;
	RTRIG_ShiftTrigger 	: R_TRIG;
	ShiftData 			: ARRAY[0..20] OF stShiftData;
	
	OvrMultiplierOld	: USINT;
	TON_OvrMultFeedback : TON;
	
	_j		  : DINT;
	fbDataRequest		: FB_DataRequest;
	RTRIG_ExecuteWriteChip : R_TRIG;
	RTRIG_ExecuteReadChip : R_TRIG;
	
	tempString1 : STRING;
	tempString2 : STRING;
	tempLayout  : STRING;

	sSrvNetID		: T_AmsNetID	:= '';(* TwinCAT TCP/IP server network address *)
	bEnable			: BOOL 			:= FALSE;(* TRUE => Enable client data exchange, FALSE => Disable *)
	bLog			: BOOL			:= FALSE;(* TRUE => Enable log message output, FALSE => Disable *)

	fbCloseAll		: FB_SocketCloseAll;
	bInitialize		: BOOL := TRUE;
	OvrMng			: FB_OvrMng;
	
	tempString	: STRING;
	tempStringPos : INT;
	
	
	tempPPString			: STRING;
	iPP						: INT;
	
	RTRIG_ProcessingDataExecute	 : R_TRIG;
	RTRIG_ProcessingDataDoneError	: R_TRIG;
	
	tTimeTemp					: TIME := T#100ms;
	TempInt						: UINT;
	tempCouth					: BOOL;
	
	RTRIG_GoodPieces			: R_TRIG;
	RTRIG_Scraped				: R_TRIG;
	RTRIG_BatchChange			: R_TRIG;
	TepmStatus					: eProductStatus;	
	
	RTRIG_UnloadFromSlide		: R_TRIG;
	RTRIG_UnloadFromLaser		: R_TRIG;
	RTRIG_UnloadFromCart		: R_TRIG;
	RTRIG_UnloadFromDeburring	: R_TRIG;
	RTRIG_UnloadFromPallet		: R_TRIG;	
	RTRIG_UnloadFromManualLoad	: R_TRIG;	
	RTRIG_IdShift		: R_TRIG;
	
	RTRIG_UnloadFromSlideAck		: R_TRIG;
	RTRIG_UnloadFromLaserAck		: R_TRIG;
	RTRIG_UnloadFromCartAck			: R_TRIG;
	RTRIG_UnloadFromDeburringAck	: R_TRIG;
	RTRIG_UnloadFromPalletAck		: R_TRIG;
	RTRIG_UnloadFromManualLoadAck	: R_TRIG;
	
	FTRIG_UnloadFromSlideAck		: F_TRIG;
	FTRIG_UnloadFromLaserAck		: F_TRIG;
	FTRIG_UnloadFromCartAck			: F_TRIG;
	FTRIG_UnloadFromDeburringAck	: F_TRIG;
	FTRIG_UnloadFromPalletAck		: F_TRIG;
	FTRIG_UnloadFromManualLoadAck	: F_TRIG;
	
	CycleTime					: DWORD;
	ProcessingHMIDataManager : FB_ButtonTrigger;
	
	fbLoadingModeSelection: FB_LoadingModeChange; 
	
	manualReq : BOOL;
	LasitManualDisable : BOOL;
	fbKillMultipleNavigationPS : FB_KillMultipleNavigationPS;
	tempDint	: ARRAY[0..3] OF DINT;
	tempReal	: ARRAY[0..3] OF REAL;
	resetManual : BOOL;
	RobotLoadOffset : ARRAY[0..EC.NUM_ROBOT_OFFSET - 1] OF DUT_XYZ_Int;
	RobotUnloadOffset : ARRAY[0..EC.NUM_ROBOT_OFFSET - 1] OF DUT_XYZ_Int;
	TON_MSSQL_UpdatePartLocationsAndProcessingDataBusy : TON;
	memReq : BOOL;
	RTRIG_MSSQL_spGetProcessingDataForHMIDone : R_TRIG;
	RTRIG_MSSQL_spGetProcessingDataForHMIExecute : R_TRIG;
	IdList	: ARRAY[0..10] OF DINT;
END_VAR

fbGetCurTaskIndex();

A_00_Init();			// Initialization

/////////INPUT//////////////////////////////////////////////////////////
A_10_EC_PN_Input();				// Profinet to Ethercat
A_11_MatManager_Input();		// Buttons-Leds exchange data	

////////////////////////////////////////////////////////////////////////
//Database();

//A_30_Laser();
A_70_DataRequest();
A_80_OvrMng();

fbLoadingModeSelection(ActualMode := G.LoadingModeActive,
					  	LoadingModeSelected:= HMI.SelectedLoadingMode,
						LS_AutoMode := HMI.General.Manuals.LS[58],
						LS_ManualMode := HMI.General.Manuals.LS[56],
						LS_SemiAutoMode:= HMI.General.Manuals.LS[57],
						PS_AutoMode => HMI.General.Manuals.PS[58],
						PS_ManualMode => HMI.General.Manuals.PS[56],
						PS_SemiAutoMode => HMI.General.Manuals.PS[57]);

PRG_Diagnostic();

/////////OUTPUT//////////////////////////////////////////////////////////
A_90_EC_PN_Output();			// Profinet to Ethercat
A_91_MatManager_Output();			// Buttons-Leds exchange data

////////////////////////////////////////////////////////////////////////

ACTION A_00_Init:
IF _TaskInfo[fbGetCurTaskIndex.index].FirstCycle THEN	// First cycle of this task
	G.Ovr_CounterValue := EC.I_Ovr_CounterValue;
	
	//PRG_MSSQL_InitConnection.Enable := TRUE;
	DB.MesReadStatusCmd := TRUE;
	
	LasitManager.Init := TRUE;
	//fbFlyPowerMarkExeManagerInit := TRUE;
ELSE
	LasitManager.Init := FALSE;
END_IF
END_ACTION

ACTION A_10_EC_PN_Input:
// EV
AL671[0] := I_Y400[0];
AL671[1] := I_Y400[1];
AL671[2] := I_Y400[2];
AL671[3] := I_Y400[3];
AL671[4] := I_Y400[4];
            
AL673[0] := I_Y400[5];
AL673[1] := I_Y400[6];
AL673[2] := I_Y400[7];
AL673[3] := I_Y400[8];
AL673[4] := I_Y400[9];
AL673[5] := I_Y400[10];

////////////////////////////////////////////////////////// Memorie R

HMI.Out.KebaEnabled := I_R2200[0].0;
G.ResetButton := CNC.vKeyboard.PS[16] OR I_R2200[0].1 OR resetManual;

//ShiftData
PRG_MSSQL_spCMD_AbortProduction.Execute 	:= I_R2200[20].2;

//// Laser
LasitManager.Execute := I_R2200[25].0 OR manualReq;
G.LasitOn			:= I_R2200[25].1;


G.MachineEmpty					:= I_R2200[40].0;
HMI.out.EnableProductionAction 	:= I_R2200[41].1;

RTRIG_UnloadFromSlide.CLK := I_R2200[42].0;
RTRIG_UnloadFromLaser.CLK := I_R2200[42].1;
RTRIG_UnloadFromCart.CLK := I_R2200[42].2;
RTRIG_UnloadFromDeburring.CLK := I_R2200[42].3;
RTRIG_UnloadFromPallet.CLK := I_R2200[42].4;
RTRIG_UnloadFromManualLoad.CLK := I_R2200[42].5;
////////////////////////////////////////////////////////// Memorie D

// WId macchina e stato pezzo
FOR _iDataPos := 1 TO CNC.NUM_DATA_POSITION+3 DO
	_dDataOff := (_iDataPos)*5;	
	MEMCPY(ADR(HMI.ShiftData[_iDataPos].FLAGP.aByte), ADR(CNC.I_D2200[_dDataOff]), SIZEOF(BYTE));
	MEMCPY(ADR(HMI.ShiftData[_iDataPos].WIDP), ADR(CNC.I_D2200[_dDataOff+1]), SIZEOF(DWORD));
END_FOR

// feedback pennetta
MEMCPY(ADR(tempDint[0]), ADR(CNC.I_D2200[100]), SIZEOF(DWORD));
tempReal[0] := TO_REAL(tempDint[0]);
HMI.Out.Probe.ActualEncoderValue := tempReal[0]/1000;

MEMCPY(ADR(tempDint[1]), ADR(CNC.I_D2200[104]), SIZEOF(DWORD));
tempReal[1] := TO_REAL(tempDint[1]);
HMI.Out.Probe.ActualProbeValue := tempReal[1]/1000;
HMI.Out.Probe.Error := CNC.I_D2200[108].0;
END_ACTION

ACTION A_11_MatManager_Input:
FC_BYTE_TO_BOOLARR(ADR(HMI.General.Manuals.LS), ADR(CNC.I_R4500[0]), SIZEOF(HMI.General.Manuals.LS));
FC_BYTE_TO_BOOLARR(ADR(HMI.St0.Manuals.LS), ADR(CNC.I_R4500[60]), SIZEOF(HMI.St0.Manuals.LS));
FC_BYTE_TO_BOOLARR(ADR(HMI.St1.Manuals.LS), ADR(CNC.I_R4500[100]), SIZEOF(HMI.St1.Manuals.LS));
FC_BYTE_TO_BOOLARR(ADR(HMI.St2.Manuals.LS), ADR(CNC.I_R4500[110]), SIZEOF(HMI.St2.Manuals.LS));
FC_BYTE_TO_BOOLARR(ADR(HMI.St3.Manuals.LS), ADR(CNC.I_R4500[120]), SIZEOF(HMI.St3.Manuals.LS));
FC_BYTE_TO_BOOLARR(ADR(HMI.St4.Manuals.LS), ADR(CNC.I_R4500[130]), SIZEOF(HMI.St4.Manuals.LS));
FC_BYTE_TO_BOOLARR(ADR(HMI.St5.Manuals.LS), ADR(CNC.I_R4500[140]), SIZEOF(HMI.St5.Manuals.LS));
FC_BYTE_TO_BOOLARR(ADR(HMI.St6.Manuals.LS), ADR(CNC.I_R4500[150]), SIZEOF(HMI.St6.Manuals.LS));
FC_BYTE_TO_BOOLARR(ADR(HMI.St7.Manuals.LS), ADR(CNC.I_R4500[160]), SIZEOF(HMI.St7.Manuals.LS));
FC_BYTE_TO_BOOLARR(ADR(HMI.St8.Manuals.LS), ADR(CNC.I_R4500[170]), SIZEOF(HMI.St8.Manuals.LS));
FC_BYTE_TO_BOOLARR(ADR(HMI.St9.Manuals.LS), ADR(CNC.I_R4500[180]), SIZEOF(HMI.St9.Manuals.LS));
FC_BYTE_TO_BOOLARR(ADR(HMI.St10.Manuals.LS), ADR(CNC.I_R4500[190]),	SIZEOF(HMI.St10.Manuals.LS));
FC_BYTE_TO_BOOLARR(ADR(HMI.St11.Manuals.LS), ADR(CNC.I_R4500[200]),	SIZEOF(HMI.St11.Manuals.LS));
FC_BYTE_TO_BOOLARR(ADR(HMI.St12.Manuals.LS), ADR(CNC.I_R4500[210]),	SIZEOF(HMI.St12.Manuals.LS));
FC_BYTE_TO_BOOLARR(ADR(HMI.St13.Manuals.LS), ADR(CNC.I_R4500[220]),	SIZEOF(HMI.St13.Manuals.LS));

//Navigation
FC_BYTE_TO_BOOLARR(ADR(HMI.In.Navigation.LS[0]), ADR(CNC.I_R4500[350]), HMI.NUM_NAVIGATION_ITEMS);

// vKeyboard
FC_BYTE_TO_BOOLARR(ADR(CNC.vKeyboard.LS), ADR(CNC.I_R3950), SIZEOF(CNC.vKeyboard.LS));

//MachineData Header
FC_BYTE_TO_BOOLARR(ADR(MachineData.aBool), ADR(CNC.I_E0000[0]), SIZEOF(MachineData.aBool));
MEMCPY(ADR(MachineData.aByte), ADR(CNC.I_E0000[10]), SIZEOF(MachineData.aByte));
MEMCPY(ADR(MachineData.aWord), ADR(CNC.I_E0000[20]), SIZEOF(MachineData.aWord));

//Safety
MEMCPY(ADR(HMI.Out.Gc1000Status), ADR(CNC.I_E0000[29]), SIZEOF(HMI.Out.Gc1000Status));
MEMCPY(ADR(HMI.Out.Doors), ADR(CNC.I_E0000[30]), SIZEOF(HMI.Out.Doors));

//Counters
MEMCPY(ADR(HMI.Out.Counters.TotalPieceGood), ADR(CNC.I_E0000[60]), SIZEOF(DWORD));
MEMCPY(ADR(HMI.Out.Counters.TotalPieceScrap), ADR(CNC.I_E0000[64]), SIZEOF(DWORD));
	
// Machine CycleTime
MEMCPY(ADR(CycleTime), ADR(CNC.I_E0000[96]), SIZEOF(CycleTime));
	
//MachineData Station	
MEMCPY(ADR(MachineData.aSt[1]), ADR(CNC.I_E0000[100]), SIZEOF(MachineData.aSt));

// Lasit - senza indirizzo MB
LasitFlyPowerMarkManager.In := (CNC.FlyPowerMarkOn = 1);	

//Richiesta dato
MEMCPY(ADR(DataRequestRead.aByte[0]), ADR(CNC.HS_read[0]), SIZEOF(BYTE));
MEMCPY(ADR(DataRequestRead.aDWord), ADR(CNC.HS_read[6]), SIZEOF(DWORD));
END_ACTION

ACTION A_30_Laser:
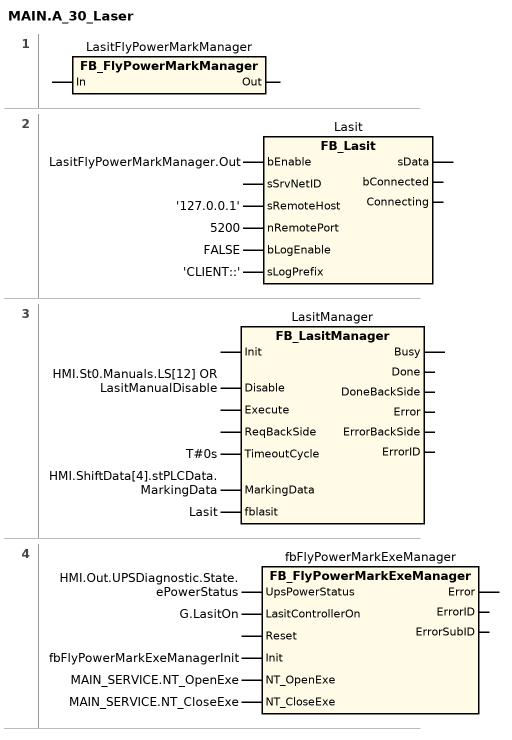
// NETWORK 1
LasitFlyPowerMarkManager(); // FB_FlyPowerMarkManager

// NETWORK 2
Lasit(
    bEnable := LasitFlyPowerMarkManager.Out,
    sRemoteHost := '127.0.0.1',
    nRemotePort := 5200,
    bLogEnable := FALSE,
    sLogPrefix := 'CLIENT::'); // FB_Lasit

// NETWORK 3
LasitManager(
    Disable := HMI.St0.Manuals.LS[12] OR LasitManualDisable,
    TimeoutCycle := T#0s,
    MarkingData := HMI.ShiftData[4].stPLCData.MarkingData,
    fblasit := Lasit); // FB_LasitManager

// NETWORK 4
fbFlyPowerMarkExeManager(
    UpsPowerStatus := HMI.Out.UPSDiagnostic.State.ePowerStatus,
    LasitControllerOn := G.LasitOn,
    Init := fbFlyPowerMarkExeManagerInit,
    NT_OpenExe := MAIN_SERVICE.NT_OpenExe,
    NT_CloseExe := MAIN_SERVICE.NT_CloseExe); // FB_FlyPowerMarkExeManager
END_ACTION

ACTION A_70_DataRequest:
fbDataRequest( ExecuteCurrent  := CNC.DataRequestRead.aByte[0].aBit.b0 OR G.RequestActual,
			   ExecuteNext	:= CNC.DataRequestRead.aByte[0].aBit.b1 OR G.RequestNext, 
			   Reset 		:= G.ResetButton,
			   WID			:= CNC.DataRequestRead.aDWord,
			   WID_Old		:= G.WID_Old,
			   MachineEmpty	:= G.MachineEmpty,
			   Done			=> CNC.DataRequestWrite.aByte[0].aBit.b0,
			   Busy			=> ,
			   Error		=> CNC.DataRequestWrite.aByte[0].aBit.b1,
			   ErrorCodePMC => CNC.DataRequestWrite.aByte[1].aByte,		 
			   St0Data 		:= St0DataTemp,
			   PMC_ShiftManData0 := HMI.ShiftData[0],
			   fbShiftDataBuffer := fbShiftDataBuffer);
			   
fbShiftDataBuffer(ArraySize := UINT_TO_INT(G.DATABUFFER_SIZE), DataRepository := ADR(G.DataBuffer));
FOR i := 1 TO NUM_STATIONS DO
	FC_DataFind(HMI.ShiftData[i].WIDP, ADR(HMI.ShiftData[i].PmcData), ADR(HMI.ShiftData[i].stPLCData), ADR(G.DataBuffer));
	IF HMI.ShiftData[i].WIDP = DB.ProcessingHMIDataLocation[i].PartId THEN	
		HMI.ShiftData[i].ProcessingData := DB.ProcessingHMIDataViewData[i];
	END_IF
END_FOR

FOR i := 0 TO NUM_STATIONS DO
	IdList[i] := HMI.ShiftData[i].WIDP;
END_FOR

IF NOT G.MachineEmpty AND MEMCMP(ADR(IdList), ADR(G.IdList_Old), SIZEOF(IdList)) <> 0 THEN
	G.UpdatePartLocationsAndProcessingDataTrigger := TRUE;
	MEMCPY(ADR(G.IdList_Old), ADR(IdList), SIZEOF(G.IdList_Old));
END_IF

//unload managment
//////////////////////Prima di rimuovere i dati dalla struttura mi salvo info per gestire tutto il resto //////////////////////
////////////////////// updateProcessingData per database, dati per oee per sapere se pezzo ok o scarto //////////////////////
////////////////////// NOTA LA POSIZIONE 17 è DOVE VENGONO SALVATI I DATI DEL PEZZO SCARICATO DAL PMC //////////////////////

IF RTRIG_UnloadFromSlide.Q THEN
	FC_UnloadManager(G.fbProcessingData[1].UnloadingStation, HMI.ShiftData[17].FLAGP);
	G.PMCShiftDataSlide := HMI.ShiftData[17];
	FC_OeeSetUpdateCount(HMI.ShiftData[17].FLAGP);
	FC_UpdatePieceCount(HMI.ShiftData[17].FLAGP, ADR(HMI.Out.Header.Pieces));
END_IF
IF RTRIG_UnloadFromLaser.Q THEN
	FC_UnloadManager(G.fbProcessingData[2].UnloadingStation, HMI.ShiftData[17].FLAGP);
	G.PMCShiftDataLaser := HMI.ShiftData[17];
	FC_OeeSetUpdateCount(HMI.ShiftData[17].FLAGP);
	FC_UpdatePieceCount(HMI.ShiftData[17].FLAGP, ADR(HMI.Out.Header.Pieces));
END_IF
IF RTRIG_UnloadFromCart.Q THEN
	FC_UnloadManager(G.fbProcessingData[5].UnloadingStation, HMI.ShiftData[17].FLAGP);
	G.PMCShiftDataCart := HMI.ShiftData[17];
	FC_OeeSetUpdateCount(HMI.ShiftData[17].FLAGP);
	FC_UpdatePieceCount(HMI.ShiftData[17].FLAGP, ADR(HMI.Out.Header.Pieces));
END_IF
IF RTRIG_UnloadFromDeburring.Q THEN
	FC_UnloadManager(G.fbProcessingData[8].UnloadingStation, HMI.ShiftData[17].FLAGP);
	G.PMCShiftDataDeburring := HMI.ShiftData[17];
	FC_OeeSetUpdateCount(HMI.ShiftData[17].FLAGP);
	FC_UpdatePieceCount(HMI.ShiftData[17].FLAGP, ADR(HMI.Out.Header.Pieces));
END_IF
IF RTRIG_UnloadFromPallet.Q THEN
	FC_UnloadManager(G.fbProcessingData[9].UnloadingStation, HMI.ShiftData[17].FLAGP);
	G.PMCShiftDataPallet := HMI.ShiftData[17];
	FC_OeeSetUpdateCount(HMI.ShiftData[17].FLAGP);
	FC_UpdatePieceCount(HMI.ShiftData[17].FLAGP, ADR(HMI.Out.Header.Pieces));
END_IF
IF RTRIG_UnloadFromManualLoad.Q THEN
	FC_UnloadManager(G.fbProcessingData[14].UnloadingStation, HMI.ShiftData[17].FLAGP);
	G.PMCShiftDataPallet := HMI.ShiftData[17];
	FC_OeeSetUpdateCount(HMI.ShiftData[17].FLAGP);
	FC_UpdatePieceCount(HMI.ShiftData[17].FLAGP, ADR(HMI.Out.Header.Pieces));	
END_IF

RTRIG_UnloadFromSlide(Q => DB.fbTriggerSequencer.In[0]);
RTRIG_UnloadFromLaser(Q => DB.fbTriggerSequencer.In[1]);
RTRIG_UnloadFromCart(Q => DB.fbTriggerSequencer.In[2]);
RTRIG_UnloadFromDeburring(Q => DB.fbTriggerSequencer.In[3]);
RTRIG_UnloadFromPallet(Q => DB.fbTriggerSequencer.In[4]);
RTRIG_UnloadFromManualLoad(Q => DB.fbTriggerSequencer.In[5]);
RTRIG_IdShift(CLK := G.UpdatePartLocationsAndProcessingDataTrigger,Q => DB.fbTriggerSequencer.In[5]);

//////////////////////////////////////////////////////////////////////////////
// dopo UpdatePartLocationAndProcessingData posso richiedere a database i ProcessingDataHMI aggiornati 	   
//RTRIG_ProcessingHMIDataExecute(CLK:= PRG_MSSQL_UpdatePartLocationsAndProcessingData.Done);
TON_MSSQL_UpdatePartLocationsAndProcessingDataBusy(IN := NOT PRG_MSSQL_UpdatePartLocationsAndProcessingData.Busy AND NOT PRG_MSSQL_UpdatePartLocationsAndProcessingData.Execute, PT := T#100MS);
ProcessingHMIDataManager(I_Command			:= (fbDataRequest.Done OR PRG_MSSQL_UpdatePartLocationsAndProcessingData.Done)
												AND NOT PRG_MSSQL_UpdatePartLocationsAndProcessingData.Execute AND NOT PRG_MSSQL_UpdatePartLocationsAndProcessingData.Busy,
                     	 I_CommandEnable	:= TRUE,	
                     	 I_Reset			:= PRG_MSSQL_spGetProcessingDataForHMI.Done OR PRG_MSSQL_spGetProcessingDataForHMI.Error,	
                     	 I_ResetEnable		:= TRUE,
						 Q_Out				:= PRG_MSSQL_spGetProcessingDataForHMI.Execute);

RTRIG_MSSQL_spGetProcessingDataForHMIDone(CLK := PRG_MSSQL_spGetProcessingDataForHMI.Done);						 
IF RTRIG_MSSQL_spGetProcessingDataForHMIDone.Q THEN
	memReq := TRUE;
END_IF

IF memReq AND NOT HMI.Out.ProductionQueueRefresh THEN
	memReq := FALSE;
END_IF
END_ACTION

ACTION A_80_OvrMng:

IF MachineData.aByte[3] <> 10 AND MachineData.aByte[3] <> 1 THEN
	OvrMng.I_Multiplier := 1;
ELSE
	OvrMng.I_Multiplier := MachineData.aByte[3];
END_IF


OvrMng(
	I_CounterValue 		:= EC.I_Ovr_CounterValue,
	I_SetCounterDone 	:= EC.I_Ovr_SetCounterDone,
	I_Overflow			:= EC.I_Ovr_Overflow,
	I_Underflow			:= EC.I_Ovr_Underflow,
	I_CounterValueOld	:= G.Ovr_CounterValue,
	I_Multiplier		:=,
	I_SetCounter		:=,
	I_SetCounterValue	:=,
	I_OvrMaxValue		:= 100,
	I_OvrMinValue		:= 0,
	Q_SetCounter 		=> EC.Q_Ovr_SetCounter,
	Q_SetCounterValue	=> EC.Q_Ovr_SetCounterValue,
	Q_Ovr				:= G.Ovr
);
END_ACTION

ACTION A_90_EC_PN_Output:
////////////////////////////////////////////////////////// Memorie R
/// allarme beckhoff ferma in fase PMC
Q_R2000[0].0 := MAIN_SERVICE.MSSQL_Events.Cumulative OR MAIN_SERVICE.Marker_Events.Cumulative OR MAIN_SERVICE.DataRequest_Events.Cumulative;

//Svuotamento forzato
CNC.Q_R2000[20].2 := PRG_MSSQL_spCMD_AbortProduction.Done;
CNC.Q_R2000[20].3 := PRG_MSSQL_spCMD_AbortProduction.Error;

//// Laser
Q_R2000[25].0 := LasitManager.Done;	
Q_R2000[25].1 := LasitManager.Error;

// Ack unload trigger
RTRIG_UnloadFromSlideAck(CLK := G.fbProcessingData[1].UnloadingStation);
RTRIG_UnloadFromLaserAck(CLK := G.fbProcessingData[2].UnloadingStation);
RTRIG_UnloadFromCartAck(CLK := G.fbProcessingData[5].UnloadingStation);
RTRIG_UnloadFromDeburringAck(CLK := G.fbProcessingData[8].UnloadingStation);
RTRIG_UnloadFromPalletAck(CLK := G.fbProcessingData[9].UnloadingStation);
RTRIG_UnloadFromManualLoadAck(CLK := G.fbProcessingData[14].UnloadingStation);

FTRIG_UnloadFromSlideAck(CLK := RTRIG_UnloadFromSlide.CLK);
FTRIG_UnloadFromLaserAck(CLK := RTRIG_UnloadFromLaser.CLK);
FTRIG_UnloadFromCartAck(CLK := RTRIG_UnloadFromCart.CLK);
FTRIG_UnloadFromDeburringAck(CLK := RTRIG_UnloadFromDeburring.CLK);
FTRIG_UnloadFromPalletAck(CLK := RTRIG_UnloadFromPallet.CLK);
FTRIG_UnloadFromManualLoadAck(CLK := RTRIG_UnloadFromManualLoad.CLK);

IF RTRIG_UnloadFromSlideAck.Q THEN 		Q_R2000[42].0 := TRUE; END_IF
IF RTRIG_UnloadFromLaserAck.Q THEN 		Q_R2000[42].1 := TRUE; END_IF
IF RTRIG_UnloadFromCartAck.Q THEN 		Q_R2000[42].2 := TRUE; END_IF
IF RTRIG_UnloadFromDeburringAck.Q THEN 	Q_R2000[42].3 := TRUE; END_IF
IF RTRIG_UnloadFromPalletAck.Q THEN 	Q_R2000[42].4 := TRUE; END_IF
IF RTRIG_UnloadFromManualLoadAck.Q THEN 	Q_R2000[42].5 := TRUE; END_IF

IF FTRIG_UnloadFromSlideAck.Q THEN 		Q_R2000[42].0 := FALSE; END_IF
IF FTRIG_UnloadFromLaserAck.Q THEN 		Q_R2000[42].1 := FALSE; END_IF
IF FTRIG_UnloadFromCartAck.Q THEN 		Q_R2000[42].2 := FALSE; END_IF
IF FTRIG_UnloadFromDeburringAck.Q THEN 	Q_R2000[42].3 := FALSE; END_IF
IF FTRIG_UnloadFromPalletAck.Q THEN 	Q_R2000[42].4 := FALSE; END_IF
IF FTRIG_UnloadFromManualLoadAck.Q THEN 	Q_R2000[42].5 := FALSE; END_IF

////////////////////////////////////////////////////////// Memorie D

//Ovr
CNC.Q_D2000[0] := G.Ovr;

//Robot load override 
CNC.Q_D2000[2] := TO_BYTE( MIN(HMI.RobotLoadSetpoint.Override, EC.NUM_MAX_ROBOT_OVR) );

//Robot unload override 
CNC.Q_D2000[3] := TO_BYTE( MIN(HMI.RobotUnloadSetpoint.Override, EC.NUM_MAX_ROBOT_OVR) );

// soglie pennetta
HMI.Out.Probe.UpperLimit := 0.1;
tempDint[2] := TO_DINT(HMI.Out.Probe.UpperLimit*1000);
MEMCPY(ADR(CNC.Q_D2000[4]), ADR(tempDint[2]), SIZEOF(DWORD));
HMI.Out.Probe.LowerLimit := -0.1;
tempDint[3] := TO_DINT(HMI.Out.Probe.LowerLimit*1000);
MEMCPY(ADR(CNC.Q_D2000[8]), ADR(tempDint[3]), SIZEOF(DWORD));

// questo serve perchè pannello fa schifo
IF HMI.St4.BroachTarget = 0 THEN HMI.St4.BroachTarget := 1; END_IF
IF HMI.St5.BroachTarget = 0 THEN HMI.St5.BroachTarget := 1; END_IF
IF HMI.St6.BroachTarget = 0 THEN HMI.St6.BroachTarget := 1; END_IF
IF HMI.St7.BroachTarget = 0 THEN HMI.St7.BroachTarget := 1; END_IF
IF HMI.St8.BroachTarget = 0 THEN HMI.St8.BroachTarget := 1; END_IF
IF HMI.St9.BroachTarget = 0 THEN HMI.St9.BroachTarget := 1; END_IF
IF HMI.St10.BroachTarget = 0 THEN HMI.St10.BroachTarget := 1; END_IF

// Broccia tagert per comando vai a
CNC.Q_D2000[20] := TO_BYTE( MAX( MIN(HMI.St4.BroachTarget,  EC.NUM_MAX_BROACH), EC.NUM_MIN_BROACH) );
CNC.Q_D2000[21] := TO_BYTE( MAX( MIN(HMI.St5.BroachTarget,  EC.NUM_MAX_BROACH), EC.NUM_MIN_BROACH) );
CNC.Q_D2000[22] := TO_BYTE( MAX( MIN(HMI.St6.BroachTarget,  EC.NUM_MAX_BROACH), EC.NUM_MIN_BROACH) );
CNC.Q_D2000[23] := TO_BYTE( MAX( MIN(HMI.St7.BroachTarget,  EC.NUM_MAX_BROACH), EC.NUM_MIN_BROACH) );
CNC.Q_D2000[24] := TO_BYTE( MAX( MIN(HMI.St8.BroachTarget,  EC.NUM_MAX_BROACH), EC.NUM_MIN_BROACH) );
CNC.Q_D2000[25] := TO_BYTE( MAX( MIN(HMI.St9.BroachTarget,  EC.NUM_MAX_BROACH), EC.NUM_MIN_BROACH) );
CNC.Q_D2000[26] := TO_BYTE( MAX( MIN(HMI.St10.BroachTarget, EC.NUM_MAX_BROACH), EC.NUM_MIN_BROACH) );

// dragante
MEMCPY(ADR(CNC.Q_D2000[28]), ADR(HMI.ChipConveyorSetpoint), SIZEOF(WORD));

// dragante
MEMCPY(ADR(CNC.Q_D2000[30]), ADR(HMI.DropsaSetpoint), SIZEOF(WORD));

//Robot load offset
FOR i := 0 TO EC.NUM_ROBOT_OFFSET - 1 DO
	RobotLoadOffset[i].X := TO_INT(HMI.RobotLoadSetpoint.PositionOffset[i].X *1000);
	RobotLoadOffset[i].Y := TO_INT(HMI.RobotLoadSetpoint.PositionOffset[i].Y *1000);
	RobotLoadOffset[i].Z := TO_INT(HMI.RobotLoadSetpoint.PositionOffset[i].Z *1000);
END_FOR
MEMCPY(ADR(CNC.Q_D2000[40]), ADR(RobotLoadOffset), SIZEOF(DUT_XYZ_Int)*EC.NUM_ROBOT_OFFSET);

//Robot unload offset
FOR i := 0 TO EC.NUM_ROBOT_OFFSET - 1 DO
	RobotUnloadOffset[i].X := TO_INT(HMI.RobotUnloadSetpoint.PositionOffset[i].X *1000);
	RobotUnloadOffset[i].Y := TO_INT(HMI.RobotUnloadSetpoint.PositionOffset[i].Y *1000);
	RobotUnloadOffset[i].Z := TO_INT(HMI.RobotUnloadSetpoint.PositionOffset[i].Z *1000);
END_FOR	
MEMCPY(ADR(CNC.Q_D2000[64]), ADR(RobotUnloadOffset), SIZEOF(DUT_XYZ_Int)*EC.NUM_ROBOT_OFFSET);
END_ACTION

ACTION A_91_MatManager_Output:
FC_BOOLARR_TO_BYTE(ADR(CNC.Q_R4000[0]), ADR(HMI.General.Manuals.PS), SIZEOF(HMI.General.Manuals.PS));
FC_BOOLARR_TO_BYTE(ADR(CNC.Q_R4000[60]), ADR(HMI.St0.Manuals.PS), SIZEOF(HMI.St0.Manuals.PS));
FC_BOOLARR_TO_BYTE(ADR(CNC.Q_R4000[100]), ADR(HMI.St1.Manuals.PS), SIZEOF(HMI.St1.Manuals.PS));
FC_BOOLARR_TO_BYTE(ADR(CNC.Q_R4000[110]), ADR(HMI.St2.Manuals.PS), SIZEOF(HMI.St2.Manuals.PS));
FC_BOOLARR_TO_BYTE(ADR(CNC.Q_R4000[120]), ADR(HMI.St3.Manuals.PS), SIZEOF(HMI.St3.Manuals.PS));
FC_BOOLARR_TO_BYTE(ADR(CNC.Q_R4000[130]), ADR(HMI.St4.Manuals.PS), SIZEOF(HMI.St4.Manuals.PS));
FC_BOOLARR_TO_BYTE(ADR(CNC.Q_R4000[140]), ADR(HMI.St5.Manuals.PS), SIZEOF(HMI.St5.Manuals.PS));
FC_BOOLARR_TO_BYTE(ADR(CNC.Q_R4000[150]), ADR(HMI.St6.Manuals.PS), SIZEOF(HMI.St6.Manuals.PS));
FC_BOOLARR_TO_BYTE(ADR(CNC.Q_R4000[160]), ADR(HMI.St7.Manuals.PS), SIZEOF(HMI.St7.Manuals.PS));
FC_BOOLARR_TO_BYTE(ADR(CNC.Q_R4000[170]), ADR(HMI.St8.Manuals.PS), SIZEOF(HMI.St8.Manuals.PS));
FC_BOOLARR_TO_BYTE(ADR(CNC.Q_R4000[180]), ADR(HMI.St9.Manuals.PS), SIZEOF(HMI.St9.Manuals.PS));
FC_BOOLARR_TO_BYTE(ADR(CNC.Q_R4000[190]), ADR(HMI.St10.Manuals.PS), SIZEOF(HMI.St10.Manuals.PS));
FC_BOOLARR_TO_BYTE(ADR(CNC.Q_R4000[200]), ADR(HMI.St11.Manuals.PS), SIZEOF(HMI.St11.Manuals.PS));
FC_BOOLARR_TO_BYTE(ADR(CNC.Q_R4000[210]), ADR(HMI.St12.Manuals.PS), SIZEOF(HMI.St12.Manuals.PS));
FC_BOOLARR_TO_BYTE(ADR(CNC.Q_R4000[220]), ADR(HMI.St13.Manuals.PS), SIZEOF(HMI.St13.Manuals.PS));

//Navigation
// funzione di sicurezza se si inchioda qualcosa a scada per problemi
fbKillMultipleNavigationPS(Ps := ADR(HMI.In.Navigation.PS[0]));
//
FC_BOOLARR_TO_BYTE(ADR(CNC.Q_R4000[350]), ADR(HMI.In.Navigation.PS[0]), HMI.NUM_NAVIGATION_ITEMS);

// vKeyboard
FC_BOOLARR_TO_BYTE(ADR(CNC.Q_R3900), ADR(CNC.vKeyboard.PS), SIZEOF(CNC.vKeyboard.PS));

//Richiesta dato
//MEMCPY(ADR(St0Data), ADR(St0DataTemp), SIZEOF(BYTE)*5);
MEMCPY(ADR(St0Data[0]), ADR(St0DataTemp.FlagP), SIZEOF(BYTE)*6);
MEMCPY(ADR(St0Data[6]), ADR(St0DataTemp.RunP), SIZEOF(DWORD));
MEMCPY(ADR(St0Data[10]), ADR(St0DataTemp.WindP), SIZEOF(DWORD)*2);
MEMCPY(ADR(St0Data[18]), ADR(St0DataTemp.Tpcy), SIZEOF(BYTE)*50);
MEMCPY(ADR(St0Data[68]), ADR(St0DataTemp.Data[1]), SIZEOF(DWORD)*93);
MEMCPY(ADR(St0Data[440]), ADR(St0DataTemp.DataB[1]), SIZEOF(DWORD)*20);
MEMCPY(ADR(St0Data[460]), ADR(St0DataTemp.DataAu[1]), SIZEOF(DWORD)*10);

MEMCPY(ADR(CNC.HS_write[0]), ADR(DataRequestWrite.aByte[0]), SIZEOF(BYTE));
MEMCPY(ADR(CNC.HS_write[1]), ADR(DataRequestWrite.aByte[1]), SIZEOF(BYTE));
MEMCPY(ADR(CNC.HS_write[9]), ADR(DataRequestWrite.aDWord), SIZEOF(DWORD));
END_ACTION

END_PROGRAM

// ---- FBs/LaserMarker - LASIT/FB_LasitManager.TcPOU
FUNCTION_BLOCK FB_LasitManager
VAR_INPUT
	Init			: BOOL;
	Disable			: BOOL;
	Execute			: BOOL;
	TimeoutCycle	: TIME;		// Tempo per timeout ciclo
END_VAR
VAR_OUTPUT
	Busy					: BOOL  := FALSE; // Ciclo di marcatura in corso
	Done					: BOOL  := FALSE; // Ciclo di marcatura terminato
	Error					: BOOL  := FALSE; 
	ErrorID					: INT 	:= 0; // -1: Timeout ciclo // 1020: Timeout caricamento layout // 1050: Timeout caricamento stringa // 1090: Marcatore in allarme 
	ErrorSubID				: INT 	:= 0;
END_VAR
VAR_IN_OUT
	MarkingData : DUT_stMarkingData;
	fblasit	: FB_Lasit;
END_VAR
VAR
	LastString			: ARRAY[1..9] OF T_MaxString;
	LastLayout			: SINT;
	i						: USINT;
	CmdIndex				: SINT;
	sCmdIndex				: T_MaxString;
	_iState					: INT 	:= -1;
	_RTRIG_Execute			: R_TRIG;
	_TON_TimeoutCycle		: TON;
	_TON_TimeoutTcpCmd		: TON;		// Timeout comando tcp (caricamento layout o testo da marcare)
	_TON_DelayBetweenCmd	: TON;		// Attesa tra l'invio di più comandi sia tcp che cablati
	JobList					: ARRAY[1..30] OF DUT_Job;
	ActualString			: ARRAY[1..9] OF T_MaxString;
	ActualIndex				: ARRAY[1..9] OF T_MaxString;
	NumberOfCmd				: USINT;
	tempLayout				: STRING(50);
END_VAR

IF Init	THEN
	M_Init();
END_IF

_TON_TimeoutCycle(IN:= Busy AND TimeoutCycle <> T#0MS, PT := TimeoutCycle);
_TON_TimeoutTcpCmd(PT := T#2S);
_TON_DelayBetweenCmd(PT := T#500MS);

IF _TON_TimeoutCycle.Q THEN
	ErrorSubID := _iState;
	_iState := 1999;
END_IF

// EXECUTE
_RTRIG_Execute(CLK := Execute);
IF _RTRIG_Execute.Q AND NOT Busy THEN
	Busy			:= TRUE;
	ErrorID			:= 0;
	ErrorSubID		:= 0;
	_TON_DelayBetweenCmd.IN := FALSE;
	
	_iState			:= 0;
ELSIF NOT Execute AND NOT Busy THEN
	Busy			:= FALSE;
	Done	:= FALSE; 
	Error	:= FALSE; 
	
	_iState			:= -1;	
END_IF

// CYCLE //////////////////////////////////////////////////////////////////////////////////////////////////////	
CASE _iState OF
	0:	
		IF Disable THEN
			_iState			:= 999;
		ELSIF NOT fblasit.bConnected THEN
			_iState			:= 1000;
		ELSE
			ActualString[1] := LEFT(MarkingData.ProfileLaser,3);
			ActualString[2] := RIGHT(MarkingData.ProfileLaser,2);
			ActualString[3] := LEFT(MarkingData.ProfileLaser,3);
			ActualString[4] := RIGHT(MarkingData.ProfileLaser,2);
				
			i := 0;
			tempLayout := 'Job_1';
			
			_iState			:= 10;
		END_IF

		
	10:
		CmdIndex := M_FindJobIndex(tempLayout);
		IF CmdIndex > 0 THEN
			_iState			:= 20;
		ELSE
			_iState			:= 1010;
		END_IF
		
	20:
		IF CmdIndex <> LastLayout THEN
			sCmdIndex := SINT_TO_STRING(CmdIndex);
			fblasit.JobChoice(I_Layout := sCmdIndex);
			_TON_TimeoutTcpCmd.IN 	:= TRUE;
			
			_iState	:= 30;	
		ELSE
			_TON_DelayBetweenCmd.IN := TRUE;
			_iState	:= 40;	
		END_IF
		
	30:
		IF fblasit.JobChoice_Done() THEN
			_TON_TimeoutTcpCmd.IN	:= FALSE;
			_TON_DelayBetweenCmd.IN := TRUE;
			LastLayout := CmdIndex;
			MEMSET(ADR(LastString), 0 , SIZEOF(LastString));
			
			_iState := 40;
		ELSIF _TON_TimeoutTcpCmd.Q THEN
			_TON_TimeoutTcpCmd.IN := FALSE;
			
			_iState		:= 1030;
		END_IF

	40:
		FOR i := 1 TO 9 DO
			IF ActualString[i] <> LastString[i] THEN
				EXIT;
			END_IF
		END_FOR
		IF _TON_DelayBetweenCmd.Q THEN
			_TON_DelayBetweenCmd.IN := FALSE;
			NumberOfCmd := 0;
			
			_iState			:= 50;
		END_IF
		
	50:		
		IF i <= 9 THEN
			FOR i := 1 TO 9 DO
				IF JobList[CmdIndex].IndexDynamicCmd[i] THEN
					ActualIndex[i] := USINT_TO_STRING(i);
					NumberOfCmd := NumberOfCmd + 1;
				ELSE
					ActualIndex[i] := '';
				END_IF
			END_FOR	

			NumberOfCmd := MIN(NumberOfCmd, 9);		
			
			_iState	:= 60;	
		ELSE
				
			_iState	:= 999;	
		END_IF
		
	60:
		fblasit.MultyDynamicCmd(I_NumberOfCmd:=  NumberOfCmd, I_Id := ActualIndex, I_Text := ActualString);
		_TON_TimeoutTcpCmd.IN 	:= TRUE;	
		
		_iState		:= 70;

	70:
		IF fblasit.DynamicCmd_Done() THEN
			LastString		:= ActualString;
			_TON_TimeoutTcpCmd.IN	:= FALSE;
	
			_iState		:= 999;
		ELSIF _TON_TimeoutTcpCmd.Q THEN
			_TON_TimeoutTcpCmd.IN := FALSE;
			
			_iState		:= 1070;
		END_IF
		
	999:
		
		Busy := FALSE;
		Done := TRUE;
		
END_CASE
	
	
// ERROR
IF (_iState > 999) THEN
	Busy			:= FALSE;
	ErrorID 		:= SEL(_TON_TimeoutCycle.Q, _iState, -1);
	Done	:= FALSE;
	Error := TRUE;
	_iState			:= -1;
END_IF

METHOD PRIVATE M_FindJobIndex : SINT
VAR_INPUT
	LayoutName 		: STRING(50);
END_VAR
VAR
	i : USINT;
END_VAR
FOR i := 1 TO 30 DO
	IF JobList[i].JobName = LayoutName THEN
		EXIT;
	END_IF
END_FOR
IF i > 30 THEN
	M_FindJobIndex := -1;
ELSE
	M_FindJobIndex := USINT_TO_SINT(JobList[i].JobIndex);
END_IF
END_METHOD

METHOD PRIVATE M_Init : BOOL
MEMSET(ADR(JobList), 0, SIZEOF(JobList));
JobList[1].JobName := 'Job_1';

//Job_1
JobList[1].JobIndex := 1;
JobList[1].IndexDynamicCmd[1] := TRUE;
JobList[1].IndexDynamicCmd[2] := TRUE;
JobList[1].IndexDynamicCmd[3] := TRUE;
JobList[1].IndexDynamicCmd[4] := TRUE;
JobList[1].IndexDynamicCmd[5] := FALSE;
JobList[1].IndexDynamicCmd[6] := FALSE;
JobList[1].IndexDynamicCmd[7] := FALSE;
JobList[1].IndexDynamicCmd[8] := FALSE;
JobList[1].IndexDynamicCmd[9] := FALSE;
JobList[1].IndexDynamicCmd[10] := FALSE;
END_METHOD

END_FUNCTION_BLOCK

// ---- FBs/LaserMarker - LASIT/FB_Lasit.TcPOU
FUNCTION_BLOCK FB_Lasit EXTENDS FB_EthDevice
VAR_OUTPUT
	Connecting				: BOOL  := FALSE; // Indica la connessione in corso, se Connecting = False e bConnected = False allora connessione in timeout
END_VAR
VAR
	sCmd					: T_MaxString;
	TON_WaitConnection		: TON;
END_VAR

SUPER^();
// TIMER
TON_WaitConnection( IN := bEnable, PT := T#10S);
Connecting := bEnable AND NOT TON_WaitConnection.Q AND NOT bConnected;

METHOD DynamicCmd : BOOL
// Description : Ask for the status of the machine
VAR_INPUT
	I_Id	: STRING;
	I_Text	: STRING;
END_VAR
VAR
	sTemp1 : STRING;
	sTemp2 : STRING;
	sTemp3 : STRING;
	sTemp4 : STRING;
	sTemp5 : STRING;
	sTemp6 : STRING;
END_VAR
sData := '';
sTemp1 := 'T';
sTemp2 := CONCAT(STX, sTemp1);
sTemp3 := CONCAT(SOH, sTemp2);
sTemp4 := CONCAT(sTemp3, I_Id);
sTemp5 := CONCAT(sTemp4, I_Text);
sTemp6 := CONCAT(sTemp5, ETX);
sCmd := CONCAT(sTemp6, EOT);
THIS^.Send(sCmd);
END_METHOD

METHOD DynamicCmd_Done : BOOL
VAR
	sTemp1 : T_MaxString;
END_VAR
IF sData = '' THEN
	DynamicCmd_Done := FALSE;
ELSE
	sTemp1 := sData;
	IF FC_Check_SOH(sTemp1) AND FC_Check_ACK(sTemp1) AND FC_Check_EOT(sTemp1) AND FC_Check_T(sTemp1) THEN
		DynamicCmd_Done := TRUE;
	ELSE
		DynamicCmd_Done := FALSE;
	END_IF
END_IF
END_METHOD

METHOD Init : BOOL
// Description : Ask for the status of the machine
VAR_INPUT
END_VAR
VAR
	sTemp1 : STRING;
	sTemp2 : STRING;
END_VAR
sData := '';
sTemp1 := 'IN';
sTemp2 := CONCAT(SOH, sTemp1);
sCmd := CONCAT(sTemp2, EOT);
sData := '';
this^.Send(sCmd);
END_METHOD

METHOD Init_Done : BOOL
VAR
	sTemp1 : T_MaxString;
END_VAR
IF sData = '' THEN
	Init_Done := FALSE;
ELSE
	sTemp1 := sData;
	IF FC_Check_SOH(sTemp1) AND FC_Check_ACK(sTemp1) AND FC_Check_EOT(sTemp1) AND FC_Check_IN(sTemp1) THEN
		Init_Done := TRUE;
	ELSE
		Init_Done := FALSE;
	END_IF
END_IF
END_METHOD

METHOD JobChoice : BOOL
// Description : Ask for the status of the machine
VAR_INPUT
	I_Layout	: STRING;
END_VAR
VAR
	sTemp1 : STRING;
	sTemp2 : STRING;
	sTemp3 : STRING;
	sTemp4 : STRING;
	sTemp5 : STRING;
END_VAR
sData := '';
sTemp1 := 'J';
sTemp2 := CONCAT(STX, sTemp1);
sTemp3 := CONCAT(SOH, sTemp2);
sTemp4 := CONCAT(sTemp3, I_Layout);
sTemp5 := CONCAT(sTemp4, ETX);
sCmd := CONCAT(sTemp5, EOT);
THIS^.Send(sCmd);
END_METHOD

METHOD JobChoice_Done : BOOL
VAR
	sTemp1 : T_MaxString;
END_VAR
IF sData = '' THEN
	JobChoice_Done := FALSE;
ELSE
	sTemp1 := sData;
	IF FC_Check_SOH(sTemp1) AND FC_Check_ACK(sTemp1) AND FC_Check_EOT(sTemp1) AND FC_Check_J(sTemp1) THEN
		JobChoice_Done := TRUE;
	ELSE
		JobChoice_Done := FALSE;
	END_IF
END_IF
END_METHOD

METHOD LastMarking : BOOL
// Description : Ask for the status of the machine
VAR_INPUT
END_VAR
VAR
	sTemp1 : STRING;
	sTemp2 : STRING;
	sTemp3 : STRING;
	sTemp4 : STRING;
END_VAR
sData := '';
sTemp1 := 'Q';
sTemp2 := CONCAT(STX, sTemp1);
sTemp3 := CONCAT(SOH, sTemp2);
sTemp4 := CONCAT(sTemp3, ETX);
sCmd := CONCAT(sTemp4, EOT);
THIS^.Send(sCmd);
END_METHOD

METHOD LastMarking_Done : BOOL
VAR_OUTPUT
	Q_nSN		: INT;
	Q_sStatus	: T_MaxString;
END_VAR
VAR
	sTemp1	: T_MaxString;
	sLeft	: T_MaxString;
	sRight	: T_MaxString;
	nPos	: INT;
	nLen	: INT;
END_VAR
Q_nSN 		:= 0;
Q_sStatus	:= '';
IF sData = '' THEN
	LastMarking_Done := FALSE;
ELSE
	sTemp1 := sData;
	IF FC_Check_SOH(sTemp1) AND FC_Check_ACK(sTemp1) AND FC_Check_EOT(sTemp1) THEN
		nPos := FIND(sTemp1,';');
		IF nPos <> 0 THEN
			nLen := LEN(sTemp1);
			sLeft := LEFT(sTemp1, nPos-1);
			Q_sStatus := RIGHT(sTemp1, nLen - nPos);
			Q_nSN := STRING_TO_INT(sLeft);
			LastMarking_Done := TRUE;
		ELSE
			LastMarking_Done := FALSE;
		END_IF
	ELSE
		LastMarking_Done := FALSE;
	END_IF
END_IF
END_METHOD

METHOD MultyDynamicCmd : BOOL
// Description : Ask for the status of the machine
VAR_INPUT
	I_NumberOfCmd : USINT; // FROM 1 TO 10
	I_Id	: ARRAY[1..9] OF T_MaxString;
	I_Text	: ARRAY[1..9] OF T_MaxString;
END_VAR
VAR
	sTemp1 : T_MaxString;
	sTemp2 : T_MaxString;
	sTemp3 : T_MaxString;
	sTemp4 : T_MaxString;
	sTemp5 : T_MaxString;
	sTemp6 : T_MaxString;
	sTemp7 : T_MaxString;
	i : USINT;
END_VAR
sData := '';
sTemp1 := CONCAT(STX, 'T0');
sTemp2 := ETX;

FOR i := 1 TO I_NumberOfCmd DO
	sTemp3 := CONCAT(sTemp1, I_Id[i]);
	sTemp4 := CONCAT(sTemp3, I_Text[i]);
	sTemp5 := CONCAT(sTemp4, sTemp2);
	sTemp6 := CONCAT(sTemp6, sTemp5);
END_FOR

sTemp7 := CONCAT(SOH, sTemp6);
sCmd := CONCAT(sTemp7, EOT);
THIS^.Send(sCmd);
END_METHOD

METHOD ReadStatus : BOOL
// Description : Ask for the status of the machine
VAR_INPUT
END_VAR
VAR
	sTemp1 : STRING;
	sTemp2 : STRING;
END_VAR
sData := '';
sTemp1 := 'K';
sTemp2 := CONCAT(SOH, sTemp1);
sCmd := CONCAT(sTemp2, EOT);
THIS^.Send(sCmd);
END_METHOD

METHOD ReadStatus_Done : BOOL
VAR_OUTPUT
	Q_wStatusWord1	: WORD;
	Q_wStatusWord2	: WORD;
END_VAR
VAR
	sTemp1	: T_MaxString;
	sLeft	: T_MaxString;
	sRight	: T_MaxString;
	nPos	: INT;
	nLen	: INT;
END_VAR
Q_wStatusWord1 := 0;
Q_wStatusWord2 := 0;
IF sData = '' THEN
	ReadStatus_Done := FALSE;
ELSE
	sTemp1 := sData;
	IF FC_Check_SOH(sTemp1) AND FC_Check_ACK(sTemp1) AND FC_Check_EOT(sTemp1) AND FC_Check_K(sTemp1) THEN
		nPos := FIND(sTemp1,',');
		IF nPos <> 0 THEN
			nLen := LEN(sTemp1);
			sLeft := LEFT(sTemp1, nPos-1);
			sRight := RIGHT(sTemp1, nLen - nPos);
			Q_wStatusWord1 := STRING_TO_WORD(sLeft);
			Q_wStatusWord2 := STRING_TO_WORD(sRight);
			ReadStatus_Done := TRUE;
		ELSE
			ReadStatus_Done := FALSE;
		END_IF
	ELSE
		ReadStatus_Done := FALSE;
	END_IF
END_IF
END_METHOD

METHOD Reset : BOOL
// Description : Ask for the status of the machine
VAR_INPUT
END_VAR
VAR
	sTemp1 : STRING;
	sTemp2 : STRING;
END_VAR
sData := '';
sTemp1 := 'R';
sTemp2 := CONCAT(SOH, sTemp1);
sCmd := CONCAT(sTemp2, EOT);
THIS^.Send(sCmd);
END_METHOD

